FUNCTION_BLOCK "Honeywell_variable_frequency_drives"   // FB29, SCL
{ S7_Optimized_Access := 'TRUE' }
VERSION : 0.1
   VAR_INPUT
      mb_addr : UInt := 255;
   END_VAR
   VAR_IN_OUT
      mb_query : "mb_query";
   END_VAR
   VAR
      sb : "mb_station_block_udt";
      read : Struct
         stw : Struct
            x24 : Bool;
            x25 : Bool;
            x26 : Bool;
            x27 : Bool;
            x28 : Bool;
            x29_control_place : Bool := FALSE;
            x30_control_place : Bool := FALSE;
            x31_control_place : Bool := TRUE;
            x16 : Bool;
            x17 : Bool;
            x18 : Bool;
            x19 : Bool;
            x20 : Bool;
            x21 : Bool;
            x22 : Bool;
            x23 : Bool;
            x08 : Bool;
            x09 : Bool;
            x10 : Bool;
            x11 : Bool;
            x12 : Bool;
            x13 : Bool;
            x14 : Bool;
            x15 : Bool;
            x00_Ready : Bool;
            x01_Running : Bool;
            x02_Counterclockwise : Bool;
            x03_Faulted : Bool;
            x04_Alarm : Bool;
            x05_AtReference : Bool;
            x06_ZeroSpeed : Bool;
            x07_FluxReady : Bool;
         END_STRUCT;
         d1_Output_Frequency : DInt;   // 0,01 Hz
         d2_Motor_Speed : DInt;   // 1 rpm
         d3_Motor_Current : DInt;   // 0,1 A
         d4_Motor_Torque : DInt;   // 0,1 %
         d5_Motor_Power : DInt;   // 0,1 %
         d6_Motor_Voltage : DInt;   // 0,1 V
         d7_DC_link_voltage : DInt;   // 1 V
         d8_Active_Fault_Code : DInt;
      END_STRUCT;
      write : Struct
         ctw : Struct
            x08 : Bool;
            x09 : Bool;
            x10 : Bool;
            x11 : Bool;
            x12 : Bool;
            x13 : Bool;
            x14 : Bool;
            x15 : Bool;
            x00 : Bool;
            x01_start : Bool := TRUE;
            x02_Reverse : Bool;
            x03_Reset_faults : Bool;
            x04 : Bool;
            x05 : Bool;
            x06 : Bool;
            x07 : Bool;
         END_STRUCT;
         __ : Word;
         speed_ref : UInt;   // 0â€¦10000 %
      END_STRUCT;
   END_VAR
BEGIN
   // Honeywell - Variable frequency drives
   // 
   // Web: https://customer.honeywell.com/resources/techlit/
   //      TechLitDocuments/62-0000s/62-0351.pdf

   "mb_station_block_header"(sb := #sb, mb_query := #mb_query);
   #mb_query.mb_addr := #mb_addr;

   #mb_query(mode := #mb_query.c.read.holding_reg,
             data_addr := 2151,
             data_ptr := #read);

   #mb_query(mode := #mb_query.c.write.holding_reg,
             data_addr := 2001,
             data_ptr := #write);

   "mb_station_block_footer"(sb := #sb, mb_query := #mb_query);
END_FUNCTION_BLOCK

// folder: Library/Modbus/Station blocks/Krohne

FUNCTION_BLOCK "Krohne_Optisonic"   // FB34, SCL
{ S7_Optimized_Access := 'TRUE' }
VERSION : 0.1
   VAR_INPUT
      mb_addr : UInt;
   END_VAR
   VAR_IN_OUT
      mb_query : "mb_query";
   END_VAR
   VAR
      sb : "mb_station_block_udt";
      data : Struct
         "Temperature process value" : Real;
         "Dynamic Viscosity at Process conditions" : Real;
         "Density Process" : Real;
         "Flow Process" : Real;
         "Velocity Process" : Real;
         "Speed of Sound" : Real;
      END_STRUCT;
   END_VAR
BEGIN
   // Krohne - Optisonic V6
   // 

   "mb_station_block_header"(sb := #sb,
                             mb_query := #mb_query);
   #mb_query.mb_addr := #mb_addr;

   #mb_query.mode := #mb_query.c.read.holding_reg;
   #mb_query(data_addr := 7050,
             data_ptr := #data);

   "mb_station_block_footer"(sb := #sb,
                             mb_query := #mb_query);
END_FUNCTION_BLOCK

FUNCTION_BLOCK "Krohne_MFC_300"   // FB100, SCL
TITLE = Krohne MFC 300
{ S7_Optimized_Access := 'TRUE' }
AUTHOR : OlaBjornli
FAMILY : modbus
VERSION : 0.1
// Coriolise flow meter
   VAR_INPUT
      mb_addr : UInt;
   END_VAR
   VAR_OUTPUT
      Temperature : Real;   // [degree C]
   END_VAR
   VAR_IN_OUT
      mb_query : "mb_query";
   END_VAR
   VAR
      sb : "mb_station_block_udt";
      read1 : Struct
         "Flow Velocity" : Real;   // [m/s]
         "Volume Flow" : Real;   // [m3/s]
         "Mass Flow" : Real;   // [kg/s]
         Temperature : Real := 273.15;   // [K]
         Density : Real;   // [kg/m3]
         Concentration_1 : Real;
         Concentration_2_or_Diagnosis_3 : Real;
         Concentration_Flow_1 : Real;
         Concentration_Flow_2 : Real;
         Diagnosis_1 : Real;
         Diagnosis_2 : Real;
         Display_Channel_1 : Real;
         Display_Channel_2 : Real;
         Operating_time : Real;   // [s]
      END_STRUCT;
      write1_settings : Struct
         Counter_1_Function : UInt;
         Counter_1_Measurement : UInt;
         Counter_2_Function : UInt;
         Counter_2_Measurement : UInt;
         Counter_3_Function : UInt;
         Counter_3_Measurement : UInt;
      END_STRUCT;
      exec_write : Bool;
   END_VAR
BEGIN
   // Krohne - MFC 300 
   // Flowmeter
   // 
   // Web: http://cdn.krohne.com/dlc/AD_MFC300_Modbus_en_091124_4000744801_R01.pdf
   //
   // #settings :
   //    Counter Function:
   //       1 = Sum Counter
   //       2 = + Counter
   //       3 = - Counter
   //       0 = Off
   //    Counter Measurement:
   //       21 = Volume Flow [m3]
   //       22 = Mass Flow [kg]
   //       27 = Concentration Flow 1
   //       28 = Concentration Flow 2

   "mb_station_block_header"(sb := #sb, mb_query := #mb_query);
   #mb_query.mb_addr := #mb_addr;

   #mb_query(mode := #mb_query.c.mode.read,
             data_addr := 30001, // 30000 + 1 (error in datasheet)
             data_ptr := #read1);
   #Temperature := #read1.Temperature - 273.15;

   // The write query isn't executing continuously in case that will damage eeprom
   IF #exec_write THEN
       #mb_query(mode := #mb_query.c.mode.write,
                 data_addr := 40001, // 40000 + 1,
                 data_ptr := #write1_settings);
       #exec_write := NOT #mb_query.Done;
   END_IF;

   "mb_station_block_footer"(sb := #sb, mb_query := #mb_query);
END_FUNCTION_BLOCK

// folder: Library/Modbus/Station blocks/Mettler

FUNCTION_BLOCK "mettler_toledo_IND560_loadTargetValue"   // FB87, SCL
{ S7_Optimized_Access := 'TRUE' }
VERSION : 0.1
   VAR_INPUT
      iValue : Real;
   END_VAR
   VAR_OUTPUT
      qDone : Bool;
   END_VAR
   VAR_IN_OUT
      "M" : "mettlerToledoInd560Udt";
      sb : "mb_station_block_udt";
   END_VAR
   VAR
      state : Int;
      old_value : Real;
      slot : USInt;
   END_VAR
   VAR CONSTANT
      NONE_AVAILABLE : USInt := 0;
   END_VAR
BEGIN
   // Load target value, for scale 1. Page 143, table B-6

   CASE #state OF

       0:  // Waiting for start.
           #qDone := false;
           #state +=
           BOOL_TO_INT(#old_value <> #iValue);

       1:  // Wait for available msg. slot
           #slot := "reqMsgSlot"(#"M".occupiedMsgSlots);
           #state += BOOL_TO_INT(#slot <> #NONE_AVAILABLE);

       2:  // #1 PLC loads floating point value first
           #"M".writeMsgSlot[#slot].cmd := 0;
           #"M".writeMsgSlot[#slot].data := #iValue;
           #state += 1;
       3:
           #state += BOOL_TO_INT(#"M".queryDone.write);

       4:  // #2 PLC sends command to set target 1 cutoff value 
           #"M".writeMsgSlot[#slot].cmd := 110;
           #state += 1;
       5:
           #state += BOOL_TO_INT(#"M".queryDone.write);

       6:  // #3 IND560 terminal sees new command, loads the value into the target
           //    and ends a return message to indicate the new target value.
           #state +=
           BOOL_TO_INT(#"M".queryDone.read
                       AND #"M".run.cmdAck[#slot] = 1
                       AND #"M".run.PF[#slot] = 13
                       AND #"M".readMsgSlot[#slot].data = #"M".writeMsgSlot[#slot].data);

       7:  // #4  PLC instructs IND560 terminal to start â€œusingâ€ new target value
           #"M".writeMsgSlot[#slot].cmd := 114;
           #state += 1;
       8:
           #state += BOOL_TO_INT(#"M".queryDone.write);

       9:  // #5 IND560 terminal sees new command
           #"M".writeMsgSlot[#slot].cmd := 0;

           #state +=
           BOOL_TO_INT(#"M".queryDone.read
                       AND #"M".run.cmdAck[#slot] = 2
                       AND #"M".run.PF[#slot] = 30
                       AND #"M".readMsgSlot[#slot].data = 0);

       ELSE: // Back to start.
           #"M".occupiedMsgSlots[#slot] := false; // Release msg. slot.
           #state := 0;
           #qDone := true;
           // The start signal should need to be set back false before next
           // exec. else the sequence will start over.
   END_CASE;
   #old_value := #iValue;

   // 
   IF #sb.out.error_comm THEN
       #state := 0;
       IF #slot <> #NONE_AVAILABLE THEN
           #"M".writeMsgSlot[#slot].cmd := 0;
           "releaseMsgSlot"(slot := #slot,
                            mem := #"M".occupiedMsgSlots);
       END_IF;
   END_IF;
END_FUNCTION_BLOCK

FUNCTION_BLOCK "mettler_toledo_IND560"   // FB88, SCL
{ S7_Optimized_Access := 'TRUE' }
VERSION : 0.1
   VAR_IN_OUT
      mb_query : "mb_query";
   END_VAR
   VAR
      mb_addr : UInt := 255;
      sb : "mb_station_block_udt";
      "M" : "mettlerToledoInd560Udt";   // Shared data
      loadTargetValue : "mettler_toledo_IND560_loadTargetValue";
      s : USInt;
   END_VAR
   VAR_TEMP
      c : Int;
   END_VAR
BEGIN
   // Mettler Toledo IND560 - Weighing Terminal

   // WARNING: This SB is just a draft and the block probably include errors !!

   // Necessary settings: ()
   // PLC -> Eth/IP - Modbus TCP -> IP-address
   // PLC -> Eth/IP - Modbus TCP -> Subnet-mask
   // PLC -> Data Format -> Byte order : standard
   // PLC -> Data Format -> Format     : Floating Point 

   // - Modbus tcp:
   //   https://bradysystems.com/wp-content/uploads/2012/10/IND560-PLC-Interface-Manual.pdf
   // - Product overview:
   //   http://www.atsackfillers.mobi/assets/ind560_ug_en_71209396_r04.pdf

   REGION Modbus
       "mb_station_block_header"(sb := #sb,
                                 mb_query := #mb_query);
       #mb_query.mb_addr := #mb_addr;

       #mb_query(mode := #mb_query.c.mode.read,
                 data_addr := 400001,
                 data_ptr := #"M".readMsgSlot,
                 Done => #"M".queryDone.read);

       #mb_query(mode := #mb_query.c.mode.write,
                 data_addr := 401026,
                 data_ptr := #"M".writeMsgSlot,
                 Done => #"M".queryDone.write);

       "mb_station_block_footer"(sb := #sb,
                                 mb_query := #mb_query);
   END_REGION

   REGION Read data-fix     
       // Extract bits in word in to a numbers.
       FOR #c := 1 TO 4 DO
           #"M".run.PF[#c].%X0 := #"M".readMsgSlot[#c].cmdRespons.FP_1;
           #"M".run.PF[#c].%X1 := #"M".readMsgSlot[#c].cmdRespons.FP_2;
           #"M".run.PF[#c].%X2 := #"M".readMsgSlot[#c].cmdRespons.FP_3;
           #"M".run.PF[#c].%X3 := #"M".readMsgSlot[#c].cmdRespons.FP_4;
           #"M".run.PF[#c].%X4 := #"M".readMsgSlot[#c].cmdRespons.FP_5;

           #"M".run.cmdAck[#c].%X0 := #"M".readMsgSlot[#c].cmdRespons.cmdAck1;
           #"M".run.cmdAck[#c].%X1 := #"M".readMsgSlot[#c].cmdRespons.cmdAck2;
       END_FOR;
   END_REGION


   #loadTargetValue(M := #"M",
                    sb := #sb);




   #"M".queryDone.write := false;
   #"M".queryDone.read := false;
END_FUNCTION_BLOCK

FUNCTION "releaseMsgSlot" : Void   // FC17, SCL
{ S7_Optimized_Access := 'TRUE' }
VERSION : 0.1
   VAR_IN_OUT
      slot : USInt;
      mem : Array[*] of Bool;
   END_VAR
   VAR_TEMP
      c : Int;
   END_VAR
BEGIN

   IF #slot <> 0 THEN
       #mem[#slot] := false;
   END_IF;
END_FUNCTION

FUNCTION "reqMsgSlot" : USInt   // FC18, SCL
{ S7_Optimized_Access := 'TRUE' }
VERSION : 0.1
   VAR_IN_OUT
      mem : Array[*] of Bool;
   END_VAR
   VAR_TEMP
      c : Int;
   END_VAR
BEGIN
   // Find first entry inside mem that is false.
   // set the entry to true and return the index. 

   #reqMsgSlot := 0;
   FOR #c := LOWER_BOUND(ARR := #mem, DIM := 1) TO
       UPPER_BOUND(ARR := #mem, DIM := 1)
   DO
       IF NOT #mem[#c] THEN
           #mem[#c] := true;
           #reqMsgSlot := INT_TO_USINT(#c);
           RETURN;
       END_IF;
   END_FOR;
END_FUNCTION

// folder: Library/Modbus/Station blocks/Ponsel mesure

FUNCTION_BLOCK "Ponsel_mesure_Conductivity_C4E"   // FB105, SCL
{ S7_Optimized_Access := 'TRUE' }
VERSION : 0.1
   VAR_INPUT
      mb_addr : UInt := 255;   // 255=broadcast
   END_VAR
   VAR_OUTPUT
      Temperature : Real;   // [degree C]
      Conductivity : Real;   // [uS/cm]
      Salinity : Real;   // [ppt]
      TDS_Kcl : Real;   // [ppm]
      measurement_ok : Bool;
   END_VAR
   VAR_IN_OUT
      mb_query : "mb_query";
   END_VAR
   VAR
      ponsel_mesure : "Ponsel_mesure";
   END_VAR
   VAR_TEMP
      start : Bool;
   END_VAR
BEGIN
   // Ponsel mesure - Conductivity_C4E

   #start := true; // Continuous measurements

   #ponsel_mesure.minimum_measurement_interval := T#1s;
   #ponsel_mesure(mb_addr := #mb_addr,
                  compensate_enable := false,
                  Measurement_ok => #measurement_ok,
                  start_measurement := #start,
                  mb_query := #mb_query);

   #Temperature := #ponsel_mesure.data1.value[0];  // [degree C]
   #Conductivity := #ponsel_mesure.data1.value[1]; // [uS/cm]
   #Salinity := #ponsel_mesure.data1.value[2];     // [ppt]
   #TDS_Kcl := #ponsel_mesure.data1.value[3];      // [ppm]
END_FUNCTION_BLOCK

FUNCTION_BLOCK "Ponsel_mesure_Dissolved_oxygen"   // FB106, SCL
{ S7_Optimized_Access := 'TRUE' }
VERSION : 0.1
   VAR_INPUT
      mb_addr : UInt := 10;   // 255=broadcast
      start : Bool := TRUE;   // (Else use start to init messurements)
      measurement_interval : Time := T#1M;
      compensate_atmospheric_pressure : Real := 1013.0;   // hPa
      compensate_salinity : Real := 0.0;   // ppm
   END_VAR
   VAR_OUTPUT
      Temperature : Real;   // [degree C]
      Oxygen_Sat : Real;   // [%]
      Oxygen_mgl : Real;   // [mg/L]
      Oxygen_ppm : Real;   // [ppm]
      measurement_ok : Bool;
      serial_number : String[32];
   END_VAR
   VAR_IN_OUT
      mb_query : "mb_query";
   END_VAR
   VAR
      ponsel_mesure : "Ponsel_mesure";
   END_VAR
   VAR_TEMP
      start_measurement : Bool;
   END_VAR
BEGIN
   // Aqualabo - Ponsel mesure
   // Dissolved oxygen (OPTOD)
   // 
   // Warning: Each pull for sensor measurement, will reduce the available 
   // life span. Please set the measurement interval to appropriate value.

   #start_measurement := #start; // #measurement_interval will define intervals.

   #ponsel_mesure.minimum_measurement_interval := #measurement_interval;
   #ponsel_mesure.compensate[1] := #compensate_atmospheric_pressure;
   #ponsel_mesure.compensate[2] := #compensate_salinity;
   #ponsel_mesure(mb_addr := #mb_addr,
                  compensate_enable := true,
                  Measurement_ok => #measurement_ok,
                  start_measurement := #start_measurement,
                  mb_query := #mb_query);

   #Temperature := #ponsel_mesure.data1.value[0]; // [degree C]
   #Oxygen_Sat := #ponsel_mesure.data1.value[1];  // [%]
   #Oxygen_mgl := #ponsel_mesure.data1.value[2];  // [mg/l]
   #Oxygen_ppm := #ponsel_mesure.data1.value[3];  // [ppm]

   #serial_number := #ponsel_mesure.data2.serial_number;
END_FUNCTION_BLOCK

// folder: Library/Modbus/Station blocks/Ponsel mesure/Misc

FUNCTION_BLOCK "ponselMessure_ChangeMbAddr"   // FB94, SCL
{ S7_Optimized_Access := 'TRUE' }
VERSION : 0.1
   VAR_INPUT
      current_addr : USInt;
      new_addr : UInt;
      exec : Bool := TRUE;
   END_VAR
   VAR_OUTPUT
      Done : Bool;
      Error : Bool;
   END_VAR
   VAR_IN_OUT
      mb_query : "mb_query";
   END_VAR
   VAR_TEMP
      d : Bool;
      "e" : Bool;
   END_VAR
BEGIN
   IF #new_addr < 1 OR #new_addr > 247
       OR #new_addr = #current_addr
   THEN
       #"e" := TRUE;
   ELSIF #exec THEN
       #mb_query(mb_addr := #current_addr,
                 mode := #mb_query.c.write.holding_reg,
                 data_addr := 16#A3,
                 Done => #d,
                 Error => #"e",
                 data_ptr := #new_addr);
   END_IF;
   #Done := #d;
   #Error := #"e";
END_FUNCTION_BLOCK

FUNCTION_BLOCK "Ponsel_mesure"   // FB107, SCL
{ S7_Optimized_Access := 'TRUE' }
VERSION : 0.1
   VAR_INPUT
      mb_addr : UInt;
      minimum_measurement_interval : Time := T#1M;
      compensate_enable : Bool;
      compensate : Array[1..2] of Real;
   END_VAR
   VAR_OUTPUT
      Measurement_ok : Bool;
   END_VAR
   VAR_IN_OUT
      mb_query : "mb_query";
      start_measurement : Bool;
   END_VAR
   VAR
      sb : "mb_station_block_udt";
      QueryCnt : UDInt;
      data1 : Struct
         value : Array[0..4] of Real;
         compensate_temperature : Real;
         compensate : Array[1..2] of Real;
         _ : Word;
         status : Array[0..4] of Struct
            x08_StmGamme0 : Bool;
            x09_StmGamme1 : Bool;
            x10_StmGamme2 : Bool;
            x11 : Bool;
            x12 : Bool;
            x13 : Bool;
            x14 : Bool;
            x15 : Bool;
            x00_Stm0 : Bool;
            x01_Stm1 : Bool;
            x02_Stm2 : Bool;
            x03_StmTemp : Bool;   // At least one parameter coefficient uses a temporary calibration standard (configuration during calibration)
            x04_StmHF : Bool;   // At least one parameter coefficient is outside calibration limits
            x05_StmCU : Bool;   // All parameter coefficients use default coefficient
            x06_StmHIST : Bool;   // All parameter coefficients use history coefficient
            x07_StmME : Bool;   // Dry weight is missing in at least one parameter coefficient (measurement under way)
         END_STRUCT;
         Compensates_3 : Real;
      END_STRUCT;
      data2 : Struct
         Description : String[30];
         serial_number : String[32];   // (addr 0x0D10)
         Software_version : Word;   // Heavy Weight: Major version and Light Weight: Minor Version.
         Hardware_version : Word;   // Heavy Weight: Major version and Light Weight: Minor Version.
      END_STRUCT;
      api : Struct
         idle : Bool;
         wait : Bool;
         interval : Time;
      END_STRUCT;
      _ : Bool;   // Internal variables bellow.
      state : Int;
      "timer" : TON_TIME;
      timer_in : Bool;
      timer_q : Bool;
      first_scan : Bool := TRUE;
      wait_time : UInt;
   END_VAR
   VAR_TEMP
      "word" : Word;
      c : Int;
      error : Bool;
      tIdle : Bool;
      pt : Time;
   END_VAR
BEGIN
   // Aqualabo - Ponsel mesure
   // Dissolved oxygen (OPTOD), Conductivity (C4E, CTZ), pH_Redox, Turbi    
   // 
   // - Warning: For the oxygen sensor each pull for sensor measurement,
   //   will use of the available life span. Please set the measurement
   //   interval to appropriate value.
   // - Continuous assign true to start_measurement, to continuous do
   //   meassurements. #minimum_measurement_interval wil still restrict
   //   the interval time.
   // - https://en.aqualabo.fr/userfiles/doc/User%20Manual%20Oxygen%20Optical%20digital%20sensor%20OPTOD.pdf

   "mb_station_block_header"(sb := #sb,
                             mb_query := #mb_query);
   #mb_query.mb_addr := #mb_addr;
   #mb_query.mode := #mb_query.c.read.holding_reg;

   #"timer"(IN := #timer_in,
          PT := #"timer".PT,
          Q => #timer_q);
   #timer_in := false;

   IF #sb.out.error_comm THEN // If communication error
       #state := 0;
       #Measurement_ok := false;
       #timer_in := true;  // Continue run the timer.
   ELSE
       CASE #state OF
           1:  // Compensate: Salinity, barometric pressure, temperature, etc.
               IF #compensate_enable THEN
                   #mb_query(mode := #mb_query.c.write.holding_reg,
                             data_addr := 16#5f,
                             data_ptr := #compensate);
                   #state += BOOL_TO_INT(#mb_query.Done);
               ELSE
                   #state += 1;
               END_IF;
           2:  // Read wait-time (Used later in state 4)
               #mb_query(data_addr := 16#A4,
                         data_ptr := #wait_time);
               #state += BOOL_TO_INT(#mb_query.Done);
           3:  // Start all meassurements.
               #"word" := 16#0f;
               #mb_query(mode := #mb_query.c.write.holding_reg,
                         data_addr := 16#01,
                         data_ptr := #"word");
               #state += BOOL_TO_INT(#mb_query.Done);
           4:  // Timer (Wait while sensor is obtaining measurements)
               #timer_in := true;
               PRESET_TIMER(TIMER := #"timer",
                            PT := MAX(IN1 := T_CONV(#wait_time),
                                      IN2 := T#1s)); // No less then 1s.
               #state += BOOL_TO_INT(#timer_q);
           5:  // Get data.
               #mb_query(data_addr := 16#0053,
                         data_ptr := #data1);
               // All measurements ok ?
               FOR #c := 0 TO 4 DO
                   #error := #error
                   OR #data1.status[#c].x00_Stm0
                   OR #data1.status[#c].x01_Stm1
                   OR #data1.status[#c].x02_Stm2;
               END_FOR;
               #Measurement_ok := NOT #error;
               IF #mb_query.Done THEN
                   // #start_measurement need to be assigned
                   // true again to start a new messurement.
                   #start_measurement := false;
                   #state := 0;
                   #QueryCnt += 1;
               END_IF;
           ELSE
               #tIdle := true;
               #timer_in := true;
               #pt := SEL(G := #api.interval = T#0s,
                          IN0 := #api.interval,
                          IN1 := #minimum_measurement_interval);
               PRESET_TIMER(PT := #pt,
                            TIMER := #"timer");

               #state := BOOL_TO_INT
               (NOT #api.wait AND // #api.wait may be set by other
                // function blocks to  halt the messurements.
                #start_measurement AND (
                (* *)#timer_q // Interval controlled
                (* *)OR #first_scan)); // At statup a messurement
               // is done as fast as possible.
       END_CASE;
   END_IF;
   // #wait is a API, for other blocks to stop the messurements,
   // #idle tells other blocks that no messurement is in progress.


   IF #sb.out.error_comm
       OR #api.idle AND NOT #api.wait
   THEN
       // Description, Serial number, sw and hw version.
       #mb_query(data_addr := 3327,
                 data_ptr := #data2);
   END_IF;

   "mb_station_block_footer"(sb := #sb,
                             mb_query := #mb_query);

   #api.idle := #tIdle;
   #api.wait := false;
   #api.interval := T#0s;
   #first_scan := false;

   (* 
   Units:
   ---------------
   value0: Temperature
                         value1:                    value2:                    value3:       
   OPTOD (oxygen)    :   Oxygen [%Sat]              Oxygen [mg/l]              Oxygen [ppm]
   Turbi             :   Nephelo turbidity [NTU]    Nephelo turbidity [FNU]    TU turbidity [mg/L]
   pH_Redox          :   pH                         Redox [mV]
   conductivity_C4E  :   Conductivity C4E [uS/cm]   Salinity [ppt]             TDS - Kcl [ppm]
   Conductivity_CTZ  :   Conductivity CTZ [mS/cm]   Salinity [g/Kg]            Conductivity CTZ [mS/cm] 
                                                                               without temperature compensation                                                                  
   OPTOD: (Dissolved oxygen)
   Compensates[1]: Atmospheric pressure [hPa], default 1013 hPa
   Compensates[2]: Salinity [ppt], default 0 ppt


   Wiring: 
   Red     Wiring diagram V+
   black   Wiring diagram V-
   Green   B+ RS-485  (Siemens A)
   White   A- RS-485  (Siemens B)
   Blue    SDI-12

   Default settings:
   Buad: 9600
   Parity: none
   Modbus address: 10


   StmX:
   000: Measurement OK
   001: Measurement OK, but out of specifications
   010: Measurement OK with INFO 1 (See datasheet)
   011: Measurement OK with INFO 2 (See datasheet)
   100: Measurement impossible, out of specifications
   101: Measurement impossible with INFO 3 (See datasheet)
   110: Measurement impossible with INFO 4 (See datasheet)
   111: measurement under way (not yet available)

   StmGamme:       
   001: measurement used range 1
   010: measurement used range 2
   011: measurement used range 3
   100: measurement used range 4

   *)
END_FUNCTION_BLOCK

// folder: Library/Modbus/Station blocks/Produal

FUNCTION_BLOCK "produal_KLH_M"   // FB42, SCL
{ S7_Optimized_Access := 'TRUE' }
VERSION : 0.1
   VAR_INPUT
      mb_addr : USInt;
   END_VAR
   VAR_OUTPUT
      temperature : Real;
      humidity : Real;
      potentiometer : Real;
   END_VAR
   VAR_IN_OUT
      mb_query : "mb_query";
   END_VAR
   VAR
      sb : "mb_station_block_udt";
      write1_calibration : Struct
         temp_offset : Int;
         humidity_offset : Int;
      END_STRUCT;
      read1 : Struct
         temperature : Int;
         humidity : UInt;
         y : Array[1..4] of UInt;
         potentiometer : Int;   // %
      END_STRUCT;
   END_VAR
BEGIN
   // Produal - KLH-M
   // Product number: 1132600
   // http://www.produal.com/shop/web_humidity_transmitters/sku-1132600

   "mb_station_block_header"(sb := #sb, mb_query := #mb_query);
   #mb_query.mb_addr := #mb_addr;

   #mb_query(mode := #mb_query.c.mode.read,
             data_addr := 30001,
             data_ptr := #read1);

   #mb_query(mode := #mb_query.c.mode.write,
             data_addr := 40006,
             data_ptr := #write1_calibration); // temp. and humidity  

   "mb_station_block_footer"(sb := #sb, mb_query := #mb_query);

   #temperature := INT_TO_REAL(#read1.temperature) * 0.1;
   #humidity := UINT_TO_REAL(#read1.humidity); // 0-100%
   #potentiometer := INT_TO_REAL(#read1.potentiometer) * 0.1;
END_FUNCTION_BLOCK

FUNCTION_BLOCK "produal_TEHR_M"   // FB43, SCL
{ S7_Optimized_Access := 'TRUE' }
VERSION : 0.1
   VAR_INPUT
      mb_addr : USInt;
      calibration_offset : Int;   // mbar
   END_VAR
   VAR_OUTPUT
      temperature : Real;   // Â°C
      analogue_output : Real;   // V
      potentiometer : Real;   // %
   END_VAR
   VAR_IN_OUT
      mb_query : "mb_query";
   END_VAR
   VAR
      sb : "mb_station_block_udt";
      r1 : Struct
         temperature : Int;
         analogue_output : UInt;
         potentiometer : Int;
      END_STRUCT;
   END_VAR
BEGIN
   // Produal - TEHR-M - Temperatur transmitter.
   // Product: 117Z190 - Pt1000 EN 60751/B
   // http://www.produal.com/shop/web_bus_temperature_transmitters/
   // sku-117Z190?hiddenAttributes_sensor_output=sensor_output_modbus&saf=true

   "mb_station_block_header"(sb := #sb,
                             mb_query := #mb_query);
   #mb_query.mb_addr := #mb_addr;

   #mb_query(mode := #mb_query.c.mode.read,
             data_addr := 30001,
             data_ptr := #r1);

   #mb_query(mode := #mb_query.c.mode.write,
             data_addr := 40001,
             data_ptr := #calibration_offset);

   "mb_station_block_footer"(sb := #sb,
                             mb_query := #mb_query);

   #temperature := INT_TO_REAL(#r1.temperature) * 0.1;
   #analogue_output := UINT_TO_REAL(#r1.analogue_output);
   #potentiometer := INT_TO_REAL(#r1.potentiometer) * 0.1;
END_FUNCTION_BLOCK

// folder: Library/Modbus/Station blocks/Scandinavian Electric

FUNCTION_BLOCK "Scandinavian_electric_CEM M-RS485"   // FB45, SCL
{ S7_Optimized_Access := 'TRUE' }
VERSION : 0.1
   VAR_INPUT
      mb_addr : UInt;
   END_VAR
   VAR_IN_OUT
      mb_query : "mb_query";
   END_VAR
   VAR
      sb : "mb_station_block_udt";
      read1 : Struct
         "Imported active energy" : UDInt;
         "Exported active energy" : UDInt;
         "Q1 Reactive energy" : UDInt;
         "Q2 Reactive energy" : UDInt;
         "Q3 Reactive energy" : UDInt;
         "Q4 Reactive energy" : UDInt;
      END_STRUCT;
      read2 : Struct
         "Partial imported active energy" : UDInt;
         "Partial exported active energy" : UDInt;
         "Q1 partial reactive energy" : UDInt;
         "Q2 partial reactive energy" : UDInt;
         "Q3 partial reactive energy" : UDInt;
         "Q4 partial reactive energy" : UDInt;
      END_STRUCT;
      serial_number : UDInt;
   END_VAR
BEGIN
   // Scandinavian Electric - Circutor - CEM M-RS485
   // Modbus interface for CEM energy meters

   // - Note: Only no parity.
   // - http://scel.no/produkter/energimaling_/_3_fase_malere/
   //   content/text_432575b2-b97f-4834-84d7-3fb83a2fdd40/1442214133237/
   //   cem_m_rs485.pdf
   // - (M014B01-03-14A)

   "mb_station_block_header"(sb := #sb, mb_query := #mb_query);
   #mb_query.mb_addr := #mb_addr;

   #mb_query.mode := #mb_query.c.read.holding_reg;
   #mb_query(data_addr := 16#0000, data_ptr := #read1);
   #mb_query(data_addr := 16#0030, data_ptr := #read2);
   #mb_query(data_addr := 16#2710, data_ptr := #serial_number);

   "mb_station_block_footer"(sb := #sb, mb_query := #mb_query);
END_FUNCTION_BLOCK

FUNCTION_BLOCK "Scandinavian_electric_Circutor_CBS"   // FB46, SCL
{ S7_Optimized_Access := 'TRUE' }
VERSION : 0.1
   VAR_INPUT
      mb_addr : UInt;
   END_VAR
   VAR_IN_OUT
      mb_query : "mb_query";
   END_VAR
   VAR
      sb : "mb_station_block_udt";
      data : Struct
         current : Array[1..8] of UInt;   // [mA]
         outputs : Array[1..8] of UInt;   // 0=Normal, 1=Pre-alarm, 2=Aktivert, 3=LÃ¥st
         pre_alarm_relay : UInt;
      END_STRUCT;
      limits : Array[1..8] of UInt;   // [mA]
   END_VAR
BEGIN
   // Scandinavian Electric - Circutor - CBS-8
   // 
   // - http://scel.no/produkter/jordfeilovervaking/
   //   varsler_panel_og_scanningsystem/content_2/
   //   text_8e3609e0-231d-4dfc-80a4-71ee43eee1af/1409662445698/cbs8.pdf

   "mb_station_block_header"(sb := #sb, mb_query := #mb_query);
   #mb_query.mb_addr := #mb_addr;

   #mb_query.mode := #mb_query.c.write.holding_reg;
   #mb_query(data_addr := 13, data_ptr := #limits);

   #mb_query.mode := #mb_query.c.read.holding_reg;
   #mb_query(data_addr := 2, data_ptr := #data);

   "mb_station_block_footer"(sb := #sb, mb_query := #mb_query);
END_FUNCTION_BLOCK

// folder: Library/Modbus/Station blocks/Schneider

FUNCTION_BLOCK "Schneider_ATV6xx"   // FB47, SCL
{ S7_Optimized_Access := 'TRUE' }
VERSION : 0.1
   VAR_INPUT
      mb_addr : USInt;
      ref_freq : Real;
   END_VAR
   VAR_IN_OUT
      mb_query : "mb_query";
   END_VAR
   VAR
      sb : "mb_station_block_udt";
      write1 : Struct
         cmd_reg : Struct
            x08_halt : Bool;
            x09 : Bool;
            x10 : Bool;
            x11_Reverse : Bool;
            x12 : Bool;
            x13 : Bool;
            x14 : Bool;
            x15 : Bool;
            x00_switch_on : Bool := TRUE;
            x01_enable_voltage : Bool := TRUE;
            x02_quick_stop : Bool;
            x03_Run : Bool;
            x04 : Bool;
            x05 : Bool;
            x06 : Bool;
            x07_fault_reset : Bool;
         END_STRUCT;
         ref_freq : Int;
      END_STRUCT;
      read1 : Struct
         status : Struct   // ETA
            x08 : Bool;
            x09_remote : Bool;   // Command or reference value via fieldbus
            x10_on_target : Bool;   // Reference value reached
            x11_ref_outside_lim : Bool;   // Reference value outside limits
            x12 : Bool;
            x13 : Bool;
            x14_stop_key : Bool;   // Manufacturer-specific Stop via STOP key
            x15_reverse : Bool;   // Manufacturer-specific
            x00_awaiting_power_stage_supply : Bool;
            x01_ready : Bool;
            x02_running : Bool;
            x03_fault : Bool;
            x04_power_stage_supply_present : Bool;
            x05_quick_stop : Bool;
            x06_power_stage_supply_disabled : Bool;
            x07_warning : Bool;
         END_STRUCT;
         output_frequency : Int;   // RFR
         frequency_reference_before_ramp : Int;   // FRH
         motor_current : Int;   // LCR
         motor_torque : Int;   // OTR
         ext_status_word : Word;
         mains_voltage : Int;   // ULN
         motor_voltage : Int;   // UOP
         drive_thermal_state : Int;   // THD
      END_STRUCT;
   END_VAR
BEGIN
   // Schneider - ATV6xx (EAV94279)
   //  
   // - http://www2.schneider-electric.com/resources/sites/SCHNEIDER_ELECTRIC/
   //   content/live/FAQS/275000/FA275868/en_US/
   //   Process%20drive%20communication%20parameters.xlsx
   // - https://profsector.com/media/catalogs/56e3af69500ef.pdf
   // - https://download.schneider-electric.com/
   //   files?p_enDocType=User+guide&p_File_Id=5470508810&
   //   p_File_Name=ATV600_EthernetIP_Modbus_TCP_Manual_EN_EAV6
   //   4328_02.pdf&p_Reference=EAV64328

   #write1.ref_freq := REAL_TO_INT(#ref_freq * 10);
   #write1.cmd_reg.x00_switch_on := #write1.cmd_reg.x03_Run := #ref_freq <> 0;

   "mb_station_block_header"(sb := #sb, mb_query := #mb_query);
   #mb_query.mb_addr := #mb_addr;

   #mb_query.mode := #mb_query.c.write.holding_reg;
   #mb_query(data_addr := 8501, data_ptr := #write1);

   #mb_query.mode := #mb_query.c.read.holding_reg;
   #mb_query(data_addr := 3201, data_ptr := #read1);

   "mb_station_block_footer"(sb := #sb, mb_query := #mb_query);
END_FUNCTION_BLOCK

FUNCTION_BLOCK "Schneider_PM556x_series"   // FB48, SCL
{ S7_Optimized_Access := 'TRUE' }
VERSION : 0.1
   VAR_INPUT
      mb_addr : UInt;
   END_VAR
   VAR_IN_OUT
      mb_query : "mb_query";
   END_VAR
   VAR
      sb : "mb_station_block_udt";
      Accumulated_Energy : Struct
         "Active Energy Delivered (Into Load)" : Real;   // kWh
         "Active Energy Received (Out of Load)" : Real;   // kWh
         "Active Energy Delivered + Received" : Real;   // kWh
         "Active Energy Delivered- Received" : Real;   // kWh
         "Reactive Energy Delivered" : Real;   // kVARh
         "Reactive Energy Received" : Real;   // kVARh
         "Reactive Energy Delivered + Received" : Real;   // kVARh
         "Reactive Energy Delivered - Received" : Real;   // kVARh
         "Apparent Energy Delivered" : Real;   // kVAh
         "Apparent Energy Received" : Real;   // kVAh
         "Apparent Energy Delivered + Received" : Real;   // kVAh
         "Apparent Energy Delivered - Received" : Real;   // kVAh
      END_STRUCT;
      data1 : Struct
         Current : Array[1..3] of Real;   // A
         "Current N" : Real;   // A
         "Current G" : Real;   // A
         "Current Avg" : Real;   // A
         "Current Unbalance" : Array[1..3] of Real;   // %
         "Current Unbalance Worst" : Real;   // %
         "Voltage L-L" : Array[1..3] of Real;   // V
         "Voltage L-L Avg" : Real;   // V
         "Voltage L-N" : Array[1..3] of Real;   // V
         "Voltage L-N Avg" : Real;   // V
         "Voltage Unbalance L-L" : Array[1..3] of Real;   // %
         "Voltage Unbalance L-L Worst" : Real;   // %
         "Voltage Unbalance L-N" : Array[1..3] of Real;   // %
         "Voltage Unbalance L-N Worst" : Real;   // %
      END_STRUCT;
      Power : Struct
         "Active Power" : Array[1..3] of Real;   // kW
         "Active Power Total" : Real;   // kW
         "Reactive Power" : Array[1..3] of Real;   // kVAR
         "Reactive Power Total" : Real;   // kVAR
         "Apparent Power" : Array[1..3] of Real;   // kVA
         "Apparent Power Total" : Real;   // kVA
         "Power Factor" : Array[1..3] of Real;   // ---
         "Power Factor Total" : Real;   // ---
         "Displacement Power Factor" : Array[1..3] of Real;   // ---
         "Displacement Power Factor Total" : Real;   // ---
      END_STRUCT;
      PF : Struct
         "Power Factor" : Array[1..3] of Real;
         "Power Factor Total" : Real;
         "Displacement Power Factor" : Array[1..3] of Real;
         "Displacement Power Factor Total" : Real;
      END_STRUCT;
      Frequency : Real;   // Hz
   END_VAR
   VAR_TEMP
      c : Int;
      t1 : Real;
      t2 : Real;
   END_VAR
BEGIN
   // Schneider Electric - PM5560, PM5563, PM5563RD
   // 
   // https://www.schneider-electric.com/en/faqs/FA234017/

   "mb_station_block_header"(sb := #sb, mb_query := #mb_query);
   #mb_query.mb_addr := #mb_addr;

   #mb_query.mode := #mb_query.c.read.holding_reg;
   #mb_query(data_addr := 2700, data_ptr := #Accumulated_Energy);
   #mb_query(data_addr := 3000, data_ptr := #data1);
   #mb_query(data_addr := 3054, data_ptr := #Power);
   #mb_query(data_addr := 3110, data_ptr := #Frequency);

   "mb_station_block_footer"(sb := #sb, mb_query := #mb_query);

   FOR #c := 1 TO 8 DO
       (* Power factor values are specially encoded floating point 
       values. Angle of complex power = power factor register value
       0° = 1, 90° = 0,  180° = -1,  270° = 2,  Q1: 0 < x < 1
       Q2: -2 < x < -1,  Q3:  -1 < x < 0,   Q4: 1 < x < 2  *)
       CASE #c OF
           1..3: #t1 := #Power."Power Factor"[#c];
           4:    #t1 := #Power."Power Factor Total";
           5..7: #t1 := #Power."Displacement Power Factor"[#c - 4];
           8:    #t1 := #Power."Displacement Power Factor Total";
       END_CASE;
       IF #t1 > 1 THEN // PF is leading
           #t2 := 2 - #t1;
       ELSIF #t1 < -1 THEN // PF is leading
           #t2 := -2 - #t1;
       ELSE            // ABS(#t1) = 1 -> PF is at unity
           #t2 := #t1; // else -> PF is lagging
       END_IF;
       CASE #c OF
           1..3: #PF."Power Factor"[#c] := #t2;
           4:    #PF."Power Factor Total" := #t2;
           5..7: #PF."Displacement Power Factor"[#c - 4] := #t2;
           8:    #PF."Displacement Power Factor Total" := #t2;
       END_CASE;
   END_FOR;
END_FUNCTION_BLOCK

FUNCTION_BLOCK "Schneider_PM1000_series"   // FB49, SCL
TITLE = Schneider Electric - PM1000 Series Power Meters
{ S7_Optimized_Access := 'TRUE' }
VERSION : 0.1
   VAR_INPUT
      mb_addr : UInt;
   END_VAR
   VAR_OUTPUT
      all : Struct
         apparent_power : Real;
         active_power : Real;
         reactive_power : Real;
         power_factor : Real;
         voltage_L_L : Real;
         voltage_L_N : Real;
         current : Real;
      END_STRUCT;
      phase : Array[1..3] of Struct
         apparent_power : Real;
         active_power : Real;
         reactive_power : Real;
         power_factor : Real;
         voltage_L_L : Real;
         voltage_L_N : Real;
         current : Real;
      END_STRUCT;
   END_VAR
   VAR_IN_OUT
      mb_query : "mb_query";
   END_VAR
   VAR
      sb : "mb_station_block_udt";
   END_VAR
   VAR_TEMP
      tAll : Struct
         apparent_power : DWord;
         active_power : DWord;
         reactive_power : DWord;
         power_factor : DWord;
         voltage_L_L : DWord;
         voltage_L_N : DWord;
         current : DWord;
      END_STRUCT;
      tPhase : Array[1..3] of Struct
         apparent_power : DWord;
         active_power : DWord;
         reactive_power : DWord;
         power_factor : DWord;
         voltage_L_L : DWord;
         voltage_L_N : DWord;
         current : DWord;
      END_STRUCT;
      c : Int;
   END_VAR
BEGIN
   // Schneider Electric - PowerLogic - PM1000 Series Power Meters
   //  - PM1200
   // 
   // http://static.schneider-electric.us/docs/Power%20Management/
   // PowerLogic%20Products/Metering/PM1200%20power%20meter/
   // PLSED309039EN_PM1000_UG.pdf

   "mb_station_block_header"(sb := #sb,
                             mb_query := #mb_query);
   #mb_query.mb_addr := #mb_addr;

   #mb_query.mode := #mb_query.c.read.holding_reg;

   #mb_query(data_addr := 3901,
             data_ptr := #tAll);
   IF #mb_query.Done THEN
       #all.apparent_power := DWORD_TO_REAL(SWAP(#tAll.apparent_power));
       #all.active_power := DWORD_TO_REAL(SWAP(#tAll.active_power));
       #all.reactive_power := DWORD_TO_REAL(SWAP(#tAll.reactive_power));
       #all.power_factor := DWORD_TO_REAL(SWAP(#tAll.power_factor));
       #all.voltage_L_L := DWORD_TO_REAL(SWAP(#tAll.voltage_L_L));
       #all.voltage_L_N := DWORD_TO_REAL(SWAP(#tAll.voltage_L_N));
       #all.current := DWORD_TO_REAL(SWAP(#tAll.current));
   END_IF;

   FOR #c := 1 TO 3 DO
       CASE #c OF
           1:
               #mb_query.data_addr := 3917;
           2:
               #mb_query.data_addr := 3931;
           3:
               #mb_query.data_addr := 3945;
       END_CASE;
       #mb_query(data_ptr := #tPhase[#c]);
       IF #mb_query.Done THEN
           #phase[#c].apparent_power := DWORD_TO_REAL(SWAP(#tPhase[#c].apparent_power));
           #phase[#c].active_power := DWORD_TO_REAL(SWAP(#tPhase[#c].active_power));
           #phase[#c].reactive_power := DWORD_TO_REAL(SWAP(#tPhase[#c].reactive_power));
           #phase[#c].power_factor := DWORD_TO_REAL(SWAP(#tPhase[#c].power_factor));
           #phase[#c].voltage_L_L := DWORD_TO_REAL(SWAP(#tPhase[#c].voltage_L_L));
           #phase[#c].voltage_L_N := DWORD_TO_REAL(SWAP(#tPhase[#c].voltage_L_N));
           #phase[#c].current := DWORD_TO_REAL(SWAP(#tPhase[#c].current));
       END_IF;
   END_FOR;

   "mb_station_block_footer"(sb := #sb,
                             mb_query := #mb_query);
END_FUNCTION_BLOCK

FUNCTION_BLOCK "Schneider_power_meter_750"   // FB50, SCL
{ S7_Optimized_Access := 'TRUE' }
VERSION : 0.1
   VAR_INPUT
      mb_addr : UInt;
   END_VAR
   VAR_IN_OUT
      mb_query : "mb_query";
   END_VAR
   VAR
      sb : "mb_station_block_udt";
      data1 : Struct
         "Real Energy, Total" : Real;   // kWh
         "Apparent Energy,Tota" : Real;   // kVAh
         "Reactive Energy,Tota" : Real;   // kVARh
         "Real Power, Total" : Real;   // kW
         "Apparent Power, Total" : Real;   // kVA
         "Reactive Power, Total" : Real;   // kVAR
         "Power Factor, Total" : Real;
         "Voltage, L-L, 3PAverage" : Real;   // Volt
         "Voltage, L-N, 3PAverage" : Real;   // Volt
         "Current, 3P Average" : Real;   // Amp
         Frequency : Real;
      END_STRUCT;
      data2 : Struct
         Current : Array[1..3] of Real;
         Current_N : Real;
      END_STRUCT;
      data3 : Struct
         Voltage_L_L : Array[1..3] of Real;   // [V] 1:L1-L2, 2:L2-L3, 3:L3-L1
         Voltage_L_N : Array[1..3] of Real;   // [V]
         "Real Power" : Array[1..3] of Real;   // kW
         "Apparent Power" : Array[1..3] of Real;   // kVA
         "Reactive Power" : Array[1..3] of Real;   // kVAR
      END_STRUCT;
   END_VAR
BEGIN
   // Schneider - Power Meter 750
   // 63230-507-201A1 - 03/2007
   // 
   // Web: https://www.ccontrols.com/support/dp/SchneiderElectricPowerMeter750.pdf

   "mb_station_block_header"(sb := #sb,
                             mb_query := #mb_query);
   #mb_query.mb_addr := #mb_addr;

   #mb_query.mode := #mb_query.c.read.holding_reg;
   #mb_query(data_addr := 1000,
             data_ptr := #data1);
   #mb_query(data_addr := 1034,
             data_ptr := #data2);
   #mb_query(data_addr := 1054,
             data_ptr := #data3);

   "mb_station_block_footer"(sb := #sb,
                             mb_query := #mb_query);
END_FUNCTION_BLOCK

FUNCTION_BLOCK "Schneider_SCADAPack_4000"   // FB51, SCL
{ S7_Optimized_Access := 'TRUE' }
VERSION : 0.1
   VAR_INPUT
      mb_addr : UInt;
   END_VAR
   VAR_IN_OUT
      mb_query : "mb_query";
   END_VAR
   VAR
      sb : "mb_station_block_udt";
      data : Array[1..3] of Int;
      setting : Array[1..3] of Int;
   END_VAR
BEGIN
   // Schneider - SCADAPack 4000 
   // Models 4012, 4032 and 4102 - Transmitters
   // 
   // Web: https://s3.amazonaws.com/cdn.freshdesk.com/data/helpdesk/
   // attachments/production/5013914262/original/
   // SCADAPack_4000_Series_Transmitters.pdf?
   // X-Amz-Algorithm=AWS4-HMAC-SHA256&X-Amz-Credential=
   // AKIAJ2JSYZ7O3I4JO6DA%2F20170919%2Fus-east-1%2Fs3%2Faws4_
   // request&X-Amz-Date=20170919T163931Z&X-Amz-Expires=300&X-Amz-
   // Signature=a206005821114e23f4a38162afdf9d14bd82209c246a378f18
   // 9af628740a1509&X-Amz-SignedHeaders=Host&response-content-type=
   // application%2Fpdf

   "mb_station_block_header"(sb := #sb, mb_query := #mb_query);
   #mb_query.mb_addr := #mb_addr;

   #mb_query.mode := #mb_query.c.mode.read;
   #mb_query(data_addr := 40116, data_ptr := #data);

   #mb_query.mode := #mb_query.c.mode.write;
   #mb_query(data_addr := 40060, data_ptr := #setting);

   "mb_station_block_footer"(sb := #sb, mb_query := #mb_query);

   (*
   Setting:

   value[1] and value[2]
   ------------------
   2 = Pascal (Pa)
   3 = kiloPascal (kPa)
   4 = megaPascal (MPa)
   5 = pounds per square inch (psi)
   6 = inches of water at 68 F
   7 = ftH2O
   8 = atm
   9 = bar
   10 = kg/cm2
   11 = g/cm2
   12 = cmHg
   13 = mmHg
   14 = torr
   15 = mH2O
   16 = cmH2O
   17 = mmH2O
   18 = inHg
   19 = mbar


   value[3]
   ------------------
   20 = degrees Celsius (ï‚°C)
   21 = degrees Fahrenheit (ï‚°F)
   22 = degrees Kelvin (K)
   23 = degrees Rankine(R)

   *)
END_FUNCTION_BLOCK

FUNCTION_BLOCK "Telemecanique_Schneider_Altivar_21_inverter"   // FB71, SCL
{ S7_Optimized_Access := 'TRUE' }
VERSION : 0.1
   VAR_INPUT
      mb_addr : UInt;
      ref : Real;
      acceleration_time : Real;
   END_VAR
   VAR_IN_OUT
      mb_query : "mb_query";
   END_VAR
   VAR
      sb : "mb_station_block_udt";
      data : Struct
         Output_current : Real;
         Voltage_DC_bus : Real;
         Output_frequency : Real;
      END_STRUCT;
      read1 : Struct   // 16#fd00
         Output_frequency : Word;
         stat : Struct
            x08 : Bool;
            x09_Reverse : Bool;
            x10_Run : Bool;
            x11_Coast_stop : Bool;
            x12_Emergency_stop : Bool;
            x13_Standby_ST_ON : Bool;   // Standby: Initialization completed, not failure stop status, not alarm stop status (MOFF, LL forced stop or forced stop due to a momentary power failure), ST=ON, and RUN=ON
            x14_Standby : Bool;   // Standby: Initialization completed, not failure stop status, and not alarm stop status (MOFF, LL forced stop or forced stop due to a momentary power failure)
            x15_Local : Bool;
            x00_Failure_FL : Bool;
            x01_Failure : Bool;
            x02_Alarm : Bool;
            x03_Main_circuit_undervoltage : Bool;
            x04_THR_2 : Bool;   // THR1: PT=set value, vL, vb, Thr - THR2: PT=0, F170, F172, F173
            x05_PI_control_OFF : Bool;
            x06_Acceleration2_deceleration2 : Bool;
            x07_DC_braking : Bool;
         END_STRUCT;
      END_STRUCT;
      read2 : Struct   // 16#fe45
         Command_mode : UInt;   // 0:Terminal board, 1:Operation panel, 2:Serial
         Setpoint_mode : UInt;   // 1 VIA, 2 VIB, 3 Operation panel, 4 Serial, 5 TB up down frequency, 255 Preset speed operation
      END_STRUCT;
      read3_alarm : Struct   // 16#fe91
         x08_Over_torque : Bool;
         x09_Cumulative_operation_hours : Bool;
         x10 : Bool;
         x11 : Bool;
         x12 : Bool;
         "x13_Main circuit_undervoltage" : Bool;   // same as MS-relay status
         x14_Decelerating_stopping : Bool;   // Related: F256 setting. At the time of the instant blackout, Forced deceleration/stop
         x15_Decelerating_stopping : Bool;   // Related: F302 setting. An automatic stop during the lower limit frequency continuance
         x00_Overcurrent : Bool;
         x01_Inverter_overload : Bool;
         x02_Motor_overload : Bool;
         x03_Overheat : Bool;
         x04_Overvoltage : Bool;
         x05_Main_circuit_undervoltage : Bool;
         x06 : Bool;
         x07_Undercurrent : Bool;
      END_STRUCT;
      read4_alarm2 : Struct   // 16#fe79
         x08 : Bool;
         x09 : Bool;
         x10 : Bool;
         x11 : Bool;
         x12 : Bool;
         x13 : Bool;
         x14 : Bool;
         x15 : Bool;
         x00_Fan_life_alarm : Bool;
         x01_Circuit_board_life : Bool;
         x02_Main_circuit_capacitor_life : Bool;
         x03_User_set_alarm : Bool;
         x04 : Bool;
         x05 : Bool;
         x06 : Bool;
         x07 : Bool;
      END_STRUCT;
      read5_trip_code : UInt;   // 16#fc90
      write1 : Struct
         cmd : Struct
            x08 : Bool;
            x09_Reverse : Bool;
            x10_Run : Bool;
            x11_Coast_stop : Bool;
            x12_Emergency_stop : Bool;
            x13_Fault_reset : Bool;
            x14_Setpoint_priority : Bool := TRUE;   // Enabled regardless of the setting of FMOD
            x15_Command_priority : Bool := TRUE;   // Enabled regardless of the setting of CMOD
            x00_Preset_speed_b0 : Bool;
            x01_Preset_speed_b1 : Bool;
            x02_Preset_speed_b2 : Bool;
            x03 : Bool;
            x04_thr2 : Bool;   // THR1 : PT=set value, vL, vb, tHr - THR2 : PT=0, F170, F172, F173
            x05_PI_control : Bool;   // 0:Normal operation, 1:PI OFF
            x06_Acceleration_deceleration_pattern_2 : Bool;   // 0: Acceleration deceleration pattern 1
            x07_DC_braking : Bool;
         END_STRUCT;
         ref : UInt;
      END_STRUCT;
      write2_comm_fault_action : UInt;
      state : USInt;
   END_VAR
   VAR_TEMP
      read6 : Struct   // 16#fe03
         Output_current : UInt;
         Voltage_DC_bus : UInt;
      END_STRUCT;
      u : UInt;
   END_VAR
BEGIN
   // Telemecanique (Schneider) - Altivar 21 inverter
   // VFD (AC-drive)

   (*
   Param:  Name:             Default:    Options:          
   F800    Baud rate         19200       0: 9600 bps, 1: 19200 bps     
   F801    Parity            Even        0: None, 1: Even, 2: Odd      
   F802    Modbus address    1           0 ... 247                     

   CMOD    2 -> Serial communication
   FMOD    4 -> Serial communication
   *)

   "mb_station_block_header"(sb := #sb, mb_query := #mb_query);
   #mb_query.mb_addr := #mb_addr;

   // ==== High priotiry queries =====
   #write1.ref := REAL_TO_UINT(#ref * 100);
   #write1.cmd.x10_Run := #ref <> 0;
   #mb_query(mode := #mb_query.c.write.holding_reg,
             data_addr := 16#fa00,
             data_ptr := #write1);

   // ==== Low priority queries =====
   CASE #state OF
       0:  // Behaviour on modbus fault
           #mb_query(mode := #mb_query.c.write.holding_reg,
                     data_addr := 16#f603,
                     data_ptr := #write2_comm_fault_action);
       1:  // Acceleration time 1  (0.1)
           #u := REAL_TO_UINT(#acceleration_time * 10);
           #mb_query(mode := #mb_query.c.write.holding_reg,
                     data_addr := 16#f603,
                     data_ptr := #u);
       2:  // Basic data, status word
           #mb_query(mode := #mb_query.c.read.holding_reg,
                     data_addr := 16#fd00,
                     data_ptr := #read1);
           IF #mb_query.Done THEN
               #data.Output_frequency :=
               UINT_TO_REAL(#read1.Output_frequency) / 100; // [%]
           END_IF;
       3:  // Where the drive take commands from: modbus or Terminal board.
           #mb_query(mode := #mb_query.c.read.holding_reg,
                     data_addr := 16#fe45,
                     data_ptr := #read2);
       4:  // Alarm word 1
           #mb_query(mode := #mb_query.c.read.holding_reg,
                     data_addr := 16#fe91,
                     data_ptr := #read3_alarm);
       5:  // Alarm word 2
           #mb_query(mode := #mb_query.c.read.holding_reg,
                     data_addr := 16#fe79,
                     data_ptr := #read4_alarm2);
       6:  // Trip code
           #mb_query(mode := #mb_query.c.read.holding_reg,
                     data_addr := 16#fc90,
                     data_ptr := #read5_trip_code);
       7:  // Other data: current, DC-bus
           #mb_query(mode := #mb_query.c.read.holding_reg,
                     data_addr := 16#fe03,
                     data_ptr := #read6);
           IF #mb_query.Done THEN
               #data.Output_current :=
               (* *)UINT_TO_REAL(#read6.Output_current) / 100; // [%]
               #data.Voltage_DC_bus :=
               (* *)UINT_TO_REAL(#read6.Voltage_DC_bus) / 100; // [%]
           END_IF;
       ELSE
           #state += 1;
   END_CASE;
   IF #sb.out.error_comm THEN
       #state := 0;
   ELSIF #mb_query.Done THEN
       #state := SEL(G := #state > 7, IN0 := #state + 1, IN1 := 0);
   END_IF;

   "mb_station_block_footer"(sb := #sb, mb_query := #mb_query);

   (* Trip codes:
   NErr     0  0  No error
   OC1      1  1  Over-current during acceleration
   OC2      2  2  Over-current during deceleration
   OC3      3  3  Over-current during constant speed operation
   OCL      4  4  Over-current in load at startup
   OCA      5  5  Short circuit in arm
   EPHI     8  8  Input phase failure
   EPHO     9  9  Output phase failure
   OP1      A 10 Overvoltage during acceleration
   OP2      B 11 Overvoltage during deceleration
   OP3      C 12 Overvoltage during constant speed operation
   OL1      D 13 Over-LOAD in inverter
   OL2      E 14 Over-LOAD in motor
   OH      10 16 Overheat trip
   E       11 17 Emergency stop
   EEP1    12 18 EEPROM fault 1 (writing error)
   EEP2    13 19 EEPROM fault 2 (reading error)
   EEP3    14 20 EEPROM fault 3 (internal fault)
   Err2    15 21 RAM fault
   Err3    16 22 ROM fault
   Err4    17 23 CPU fault
   Err5    18 24 Communication error trip
   Err7    1A 26 Current detector fault
   Err8    1B 27 Optional circuit board type error
   UC      1D 29 Small-current trip
   UP1     1E 30 Trip due to undervoltage in main circuit
   Ot      20 32 Over-torque trip
   EF2     22 34 Ground fault trip (hardware detection)
   OC1P    25 37 Overcurrent flowing in element during acceleration
   OC2P    26 38 Overcurrent flowing in element during deceleration
   OC3P    27 39 Overcurrent flowing in element during operation
   EtYP    29 41 Inverter type error
   OH2     2E 46 External thermal input
   SOUt    2F 47 VIA cable break
   E-18    32 50 Break in an analog signal cable
   E-19    33 51 CPU fault
   E-20    34 52 Excess torque boost
   E-21    35 53 CPU fault
   Etn1    54 84 Auto-tuning error
   *)
END_FUNCTION_BLOCK

FUNCTION_BLOCK "Schneider_conzerv_EM6430"   // FB91, SCL
{ S7_Optimized_Access := 'TRUE' }
VERSION : 0.1
   VAR_INPUT
      mb_addr : USInt;
   END_VAR
   VAR_IN_OUT
      mb_query : "mb_query";
   END_VAR
   VAR
      sb : "mb_station_block_udt";
      read1_common : Struct
         Apparent_power_total : Real;
         Active_power_total : Real;
         Reactive_power_total : Real;
         Power_factor_average : Real;
         Voltage_average_phase_phase : Real;
         Voltage_average_phase_neutral : Real;
         Current_average : Real;
         Frequency : Real;   // Hz
      END_STRUCT;
      read2_phase : Array[1..3] of Struct
         Apparent_power : Real;
         Active_power : Real;
         Reactive_power : Real;
         Power_factor : Real;
         Voltage_phase_phase : Real;
         Voltage_phase_neutral : Real;
         Current : Real;
      END_STRUCT;
      read3_THD : Struct
         Voltage_THD : Array[1..3] of Real;
         Current_THD : Array[1..3] of Real;
      END_STRUCT;
      read4 : Struct
         Forward_apparent_energy : Real;
         Forward_active_energy : Real;
         Forward_reactive_inductive_energy : Real;
         Forward_reactive_capacitive_energy : Real;
         Reverse_apparent_energy : Real;
         Reverse_active_energy : Real;
         Reverse_reactive_inductive_Energy : Real;
         Reverse_reactive_capacitive_Energy : Real;
         Average_load_percentage : Real;
         Percentage_of_phase_load : Array[1..3] of Real;
         "Unbalanced_%load" : Real;
         "Unbalanced_%_voltage" : Real;
      END_STRUCT;
      read5_common_RMS : Struct
         Apparent_power_total : Real;
         Active_power_total : Real;
         Reactive_power_total : Real;
         Power_factor_average : Real;
         Voltage_average_phase_phase : Real;
         Voltage_average_phase_neutral : Real;
         Current_average : Real;
         Frequency : Real;   // Hz
         _ : UDInt;   // Reserved
         Number_of_interruption : UDInt;
      END_STRUCT;
   END_VAR
BEGIN
   // Schneider-electric - Conzerv EM6430 - Power meters
   // NHA12535-03
   // 
   // https://www.schneider-electric.com/resources/sites/SCHNEIDER_ELECTRIC/
   // content/live/FAQS/276000/FA276938/en_US/EM6430_User_Manual_NHA12535-03.pdf

   "mb_station_block_header"(sb := #sb, mb_query := #mb_query);
   #mb_query.mb_addr := #mb_addr; // Device address.

   #mb_query.mode := #mb_query.c.read.holding_reg;
   #mb_query(data_addr := 3901, data_ptr := #read1_common);
   #mb_query(data_addr := 3917, data_ptr := #read2_phase);
   #mb_query(data_addr := 3861, data_ptr := #read3_THD);
   #mb_query(data_addr := 3959, data_ptr := #read4);
   #mb_query(data_addr := 3001, data_ptr := #read5_common_RMS);

   "mb_station_block_footer"(sb := #sb, mb_query := #mb_query);
END_FUNCTION_BLOCK

FUNCTION_BLOCK "Schneider_PM750"   // FB92, SCL
{ S7_Optimized_Access := 'TRUE' }
VERSION : 0.1
   VAR_INPUT
      mb_addr : UInt;
   END_VAR
   VAR_IN_OUT
      mb_query : "mb_query";
   END_VAR
   VAR
      sb : "mb_station_block_udt";
      data1 : Struct
         "Real Energy, Total" : Real;   // kWh
         "Apparent Energy,Tota" : Real;   // kVAh
         "Reactive Energy,Tota" : Real;   // kVARh
         "Real Power, Total" : Real;   // kW
         "Apparent Power, Total" : Real;   // kVA
         "Reactive Power, Total" : Real;   // kVAR
         "Power Factor, Total" : Real;
         "Voltage, L-L, 3PAverage" : Real;   // Volt
         "Voltage, L-N, 3PAverage" : Real;   // Volt
         "Current, 3P Average" : Real;   // Amp
         Frequency : Real;
      END_STRUCT;
      data2 : Struct
         Current : Array[1..3] of Real;
         Current_N : Real;
      END_STRUCT;
      data3 : Struct
         Voltage_L_L : Array[1..3] of Real;   // [V] 1:L1-L2, 2:L2-L3, 3:L3-L1
         Voltage_L_N : Array[1..3] of Real;   // [V]
         "Real Power" : Array[1..3] of Real;   // kW
         "Apparent Power" : Array[1..3] of Real;   // kVA
         "Reactive Power" : Array[1..3] of Real;   // kVAR
      END_STRUCT;
   END_VAR
BEGIN
   // Schneider - Power Meter 750
   // 63230-507-201A1 - 03/2007
   // 
   // Web: https://www.ccontrols.com/support/dp/SchneiderElectricPowerMeter750.pdf

   "mb_station_block_header"(sb := #sb, mb_query := #mb_query);
   #mb_query.mb_addr := #mb_addr;

   #mb_query.mode := #mb_query.c.read.holding_reg;
   #mb_query(data_addr := 1000, data_ptr := #data1);
   #mb_query(data_addr := 1034, data_ptr := #data2);
   #mb_query(data_addr := 1054, data_ptr := #data3);

   "mb_station_block_footer"(sb := #sb, mb_query := #mb_query);
END_FUNCTION_BLOCK

// folder: Library/Modbus/Station blocks/Siemens

FUNCTION_BLOCK "siemens_PAC3200"   // FB8, SCL
{ S7_Optimized_Access := 'TRUE' }
VERSION : 0.1
   VAR_INPUT
      mb_addr : USInt := 1;
   END_VAR
   VAR_IN_OUT
      mb_query : "mb_query";
   END_VAR
   VAR
      sb : "mb_station_block_udt";
      read1 : Struct
         voltage_L_n : Array[1..3] of Real;
         "voltage _L_L" : Array[1..3] of Real;   // 1:Va-b, 2:Vb-c, 3:Vc-a,
         current : Array[1..3] of Real;
         apparent_power : Array[1..3] of Real;
         active_power : Array[1..3] of Real;
         reactive_power : Array[1..3] of Real;
         power_factor : Array[1..3] of Real;
         THD_R_voltage : Array[1..3] of Real;
      END_STRUCT;
      read2 : Struct
         frequency : Real;   // unit: hz
         avg_voltage_Vph_n : Real;   // unit: V
         avg_voltage_Vph_ph : Real;   // unit: V
         avg_current : Real;   // unit: A
         total_apparent_power : Real;   // unit: VA
         total_active_power : Real;   // unit: W
      END_STRUCT;
      read3 : Struct
         serial_number : String[16];
      END_STRUCT;
   END_VAR
BEGIN
   // - Siemens - PAC3200 - Power meter
   // - http://w3.siemens.com.br/buildingtechnologies/br/
   //   documents/manual-sentron-pac3200.pdf
   //   3.9.3, page 40

   "mb_station_block_header"(sb := #sb, mb_query := #mb_query);
   #mb_query.mb_addr := #mb_addr; // Device address.

   // Tree queries, reading one section of holding registers each.
   #mb_query.mode := #mb_query.c.read.holding_reg;
   #mb_query(data_addr := 1, data_ptr := #read1);
   #mb_query(data_addr := 55, data_ptr := #read2);
   #mb_query(data_addr := 64012, data_ptr := #read3);

   // - Each query reading one section of holding registers.
   // - Data length is automatically calculated for holding and
   //   input regisers.

   "mb_station_block_footer"(sb := #sb, mb_query := #mb_query);
END_FUNCTION_BLOCK

FUNCTION_BLOCK "Siemens_7SR11_7SR12_argus"   // FB53, SCL
{ S7_Optimized_Access := 'TRUE' }
VERSION : 0.1
   VAR_INPUT
      mb_addr : USInt := 1;
   END_VAR
   VAR_OUTPUT
      out1 : Struct
         primary_Voltage_L_L : Array[1..3] of Real;
         primary_Voltage_L_N : Array[1..3] of Real;
         secondary_Voltage_L_N : Array[1..3] of Real;
      END_STRUCT;
      out2 : Struct
         nominal_voltage_degrees_L_L : Array[1..3] of Real;
         nominal_voltage_degrees_L_N : Array[1..3] of Real;
         Vzps : Real;
         Vpps : Real;
         Vnps : Real;
         Vzps_degree : Real;
         Vpps_degree : Real;
         Vnps_degree : Real;
         frequency : Real;
      END_STRUCT;
      out3 : Struct
         primary_current : Array[1..3] of Real;
         secondary_current : Array[1..3] of Real;
         nominal_current : Array[1..3] of Real;
         nominal_current_degrees : Array[1..3] of Real;
         primary_In : Real;
         secondary_In : Real;
         nominal_In : Real;
         primary_Ig : Real;
         secondary_Ig : Real;
         nominal_Ig : Real;
         nominal_Izps : Real;
         nominal_Ipps : Real;
         nominal_Inps : Real;
         nominal_Izps_degrees : Real;
         nominal_Ipps_degrees : Real;
         nominal_Inps_degrees : Real;
      END_STRUCT;
      out4 : Struct
         active_power : Array[1..3] of Real;
         active_power_tot : Real;
         reactive_power : Array[1..3] of Real;
         reactive_power_tot : Real;
         apparent_power : Array[1..3] of Real;
         apparent_power_tot : Real;
         power_factor : Array[1..3] of Real;
         power_factor_tot : Real;
      END_STRUCT;
   END_VAR
   VAR_IN_OUT
      mb_query : "mb_query";
   END_VAR
   VAR
      sb : "mb_station_block_udt";
      out5 : Struct
         act_energy_exp : UDInt;
         act_energy_imp : UDInt;
         react_energy_exp : UDInt;
         react_energy_imp : UDInt;
         thermal_status_Ph_A : UInt;
         thermal_status_Ph_B : UInt;
         thermal_Status_Ph_C : UInt;
      END_STRUCT;
      out6 : Struct
         fault_records : Real;
         event_records : Real;
         waveform_records : Real;
         secondary_voltage : Array[1..3] of Real;
      END_STRUCT;
   END_VAR
   VAR_TEMP
      c : Int;
      read1 : Struct
         primary_Voltage_L_L : Array[1..3] of UDInt;
         primary_Voltage_L_N : Array[1..3] of UDInt;
         secondary_Voltage_L_N : Array[1..3] of UDInt;
      END_STRUCT;
      read2 : Struct
         nominal_voltage_degrees_L_L : Array[1..3] of UDInt;
         nominal_voltage_degrees_L_N : Array[1..3] of UDInt;
         Vzps : UDInt;
         Vpps : UDInt;
         Vnps : UDInt;
         Vzps_degree : UDInt;
         Vpps_degree : UDInt;
         Vnps_degree : UDInt;
         frequency : UDInt;
      END_STRUCT;
      read3 : Struct
         primary_current : Array[1..3] of UDInt;
         secondary_current : Array[1..3] of UDInt;
         nominal_current : Array[1..3] of UDInt;
         nominal_current_degrees : Array[1..3] of UDInt;
         primary_In : UDInt;
         secondary_In : UDInt;
         nominal_In : UDInt;
         primary_Ig : UDInt;
         secondary_Ig : UDInt;
         nominal_Ig : UDInt;
         nominal_Izps : UDInt;
         nominal_Ipps : UDInt;
         nominal_Inps : UDInt;
         nominal_Izps_degrees : UDInt;
         nominal_Ipps_degrees : UDInt;
         nominal_Inps_degrees : UDInt;
      END_STRUCT;
      read4 : Struct
         active_power : Array[1..3] of UDInt;
         active_power_tot : UDInt;
         reactive_power : Array[1..3] of UDInt;
         reactive_power_tot : UDInt;
         apparent_power : Array[1..3] of UDInt;
         apparent_power_tot : UDInt;
         power_factor : Array[1..3] of UDInt;
         power_factor_tot : UDInt;
      END_STRUCT;
      read6 : Struct
         fault_records : UDInt;
         event_records : UDInt;
         waveform_Records : UDInt;
         secondary_voltage : Array[1..3] of UDInt;
      END_STRUCT;
   END_VAR
BEGIN
   // Siemens - 7SR11 & 7SR12 - Argus - Overcurrent Relay
   // Energy Management
   //  
   // - https://cache.industry.siemens.com/dl/files/284/109747284/
   //   att_928907/v1/7SR12_Argus_Complete_Technical_Manual.pdf
   //   ==> page 212  

   "mb_station_block_header"(sb := #sb,
                             mb_query := #mb_query);
   #mb_query.mb_addr := #mb_addr;

   #mb_query.mode := #mb_query.c.mode.read;

   #mb_query(data_addr := 40010,
             data_ptr := #read1);
   IF #mb_query.Done THEN
       FOR #c := 1 TO 3 DO
           #out1.primary_Voltage_L_L[#c] := UDINT_TO_REAL(#read1.primary_Voltage_L_L[#c]) / 1000;
           #out1.primary_Voltage_L_N[#c] := UDINT_TO_REAL(#read1.primary_Voltage_L_N[#c]) / 1000;
           #out1.secondary_Voltage_L_N[#c] := UDINT_TO_REAL(#read1.secondary_Voltage_L_N[#c]) / 1000;
       END_FOR;
   END_IF;

   #mb_query(data_addr := 40034,
             data_ptr := #read2);
   IF #mb_query.Done THEN
       FOR #c := 1 TO 3 DO
           #out2.nominal_voltage_degrees_L_L[#c] := UDINT_TO_REAL(#read2.nominal_voltage_degrees_L_L[#c]) / 1000;
           #out2.nominal_voltage_degrees_L_N[#c] := UDINT_TO_REAL(#read2.nominal_voltage_degrees_L_N[#c]) / 1000;
       END_FOR;
       #out2.Vzps := UDINT_TO_REAL(#read2.Vzps) / 1000;
       #out2.Vpps := UDINT_TO_REAL(#read2.Vpps) / 1000;
       #out2.Vnps := UDINT_TO_REAL(#read2.Vnps) / 1000;
       #out2.Vzps_degree := UDINT_TO_REAL(#read2.Vzps_degree) / 1000;
       #out2.Vpps_degree := UDINT_TO_REAL(#read2.Vpps_degree) / 1000;
       #out2.Vnps_degree := UDINT_TO_REAL(#read2.Vnps_degree) / 1000;
       #out2.frequency := UDINT_TO_REAL(#read2.frequency) / 1000;
   END_IF;

   #mb_query(data_addr := 40064,
             data_ptr := #read3);
   IF #mb_query.Done THEN
       FOR #c := 1 TO 3 DO
           #out3.primary_current[#c] := UDINT_TO_REAL(#read3.primary_current[#c]) / 1000;
           #out3.secondary_current[#c] := UDINT_TO_REAL(#read3.secondary_current[#c]) / 1000;
           #out3.nominal_current[#c] := UDINT_TO_REAL(#read3.nominal_current[#c]) / 1000;
           #out3.nominal_current_degrees[#c] := UDINT_TO_REAL(#read3.nominal_current_degrees[#c]) / 1000;
       END_FOR;
       #out3.primary_In := UDINT_TO_REAL(#read3.primary_In) / 1000;
       #out3.secondary_In := UDINT_TO_REAL(#read3.secondary_In) / 1000;
       #out3.nominal_In := UDINT_TO_REAL(#read3.nominal_In) / 1000;
       #out3.primary_Ig := UDINT_TO_REAL(#read3.primary_Ig) / 1000;
       #out3.secondary_Ig := UDINT_TO_REAL(#read3.secondary_Ig) / 1000;
       #out3.nominal_Ig := UDINT_TO_REAL(#read3.nominal_Ig) / 1000;
       #out3.nominal_Izps := UDINT_TO_REAL(#read3.nominal_Izps) / 1000;
       #out3.nominal_Ipps := UDINT_TO_REAL(#read3.nominal_Ipps) / 1000;
       #out3.nominal_Inps := UDINT_TO_REAL(#read3.nominal_Inps) / 1000;
       #out3.nominal_Izps_degrees := UDINT_TO_REAL(#read3.nominal_Izps_degrees) / 1000;
       #out3.nominal_Ipps_degrees := UDINT_TO_REAL(#read3.nominal_Ipps_degrees) / 1000;
       #out3.nominal_Inps_degrees := UDINT_TO_REAL(#read3.nominal_Inps_degrees) / 1000;
   END_IF;

   #mb_query(data_addr := 40112,
             data_ptr := #read4);
   IF #mb_query.Done THEN
       FOR #c := 1 TO 3 DO
           #out4.active_power[#c] := UDINT_TO_REAL(#read4.active_power[#c]) / 1000;
           #out4.reactive_power[#c] := UDINT_TO_REAL(#read4.reactive_power[#c]) / 1000;
           #out4.apparent_power[#c] := UDINT_TO_REAL(#read4.apparent_power[#c]) / 1000;
           #out4.power_factor[#c] := UDINT_TO_REAL(#read4.power_factor[#c]) / 1000;
       END_FOR;
       #out4.active_power_tot := UDINT_TO_REAL(#read4.active_power_tot) / 1000;
       #out4.reactive_power_tot := UDINT_TO_REAL(#read4.reactive_power_tot) / 1000;
       #out4.apparent_power_tot := UDINT_TO_REAL(#read4.apparent_power_tot) / 1000;
       #out4.power_factor_tot := UDINT_TO_REAL(#read4.power_factor_tot) / 1000;
   END_IF;

   #mb_query(data_addr := 40144,
             data_ptr := #out5);

   #mb_query(data_addr := 40167,
             data_ptr := #read6);
   IF #mb_query.Done THEN
       FOR #c := 1 TO 3 DO
           #out6.secondary_voltage[#c] := UDINT_TO_REAL(#read6.secondary_voltage[#c]) / 1000;
       END_FOR;
       #out6.fault_records := UDINT_TO_REAL(#read6.fault_records) / 1000;
       #out6.event_records := UDINT_TO_REAL(#read6.event_records) / 1000;
       #out6.waveform_records := UDINT_TO_REAL(#read6.waveform_Records) / 1000;
   END_IF;

   "mb_station_block_footer"(sb := #sb,
                             mb_query := #mb_query);
END_FUNCTION_BLOCK

FUNCTION_BLOCK "Siemens_MAG_6000"   // FB54, SCL
{ S7_Optimized_Access := 'TRUE' }
VERSION : 0.1
   VAR_INPUT
      mb_addr : UInt;
   END_VAR
   VAR_IN_OUT
      mb_query : "mb_query";
   END_VAR
   VAR
      sb : "mb_station_block_udt";
      flow : Struct
         velocity : Real;   // mm/s
         flow : Real;
      END_STRUCT;
      totalizer : Array[1..3] of UDInt;
   END_VAR
BEGIN
   // Siemens - SITRANS F M MAG 6000

   "mb_station_block_header"(sb := #sb, mb_query := #mb_query);
   #mb_query.mb_addr := #mb_addr;

   #mb_query.mode := #mb_query.c.read.holding_reg;
   #mb_query(data_addr := 2999, data_ptr := #flow);
   #mb_query(data_addr := 3016, data_ptr := #totalizer);

   "mb_station_block_footer"(sb := #sb, mb_query := #mb_query);
END_FUNCTION_BLOCK

FUNCTION_BLOCK "Siemens_MASS_6000"   // FB55, SCL
{ S7_Optimized_Access := 'TRUE' }
VERSION : 0.1
   VAR_INPUT
      mb_addr : UInt;
   END_VAR
   VAR_IN_OUT
      mb_query : "mb_query";
   END_VAR
   VAR
      sb : "mb_station_block_udt";
      flow : Struct
         massflow : Real;   // [kg/s]
         volumeflow : Real;   // [m3/s]
         density : Real;   // [kg/m3]
         temperature : Real;   // [Â°C]
         fraction : Array[1..2] of Real;   // [kg/s]
         "%_fraction" : Real;   // [%]
         totalizer_1 : Array[1..2] of UDInt;   // [kg or m3]
         totalizer_2 : Array[1..2] of UDInt;   // [kg or m3]
         totalizer_real : Array[1..2] of Real;   // [kg or m3]
      END_STRUCT;
   END_VAR
BEGIN
   // Siemens - MASS 6000
   // https://cache.industry.siemens.com/dl/files/906/44880906/
   // att_70364/v1/USMII_MODBUS_AOM_OI_En_en-US.pdf

   "mb_station_block_header"(sb := #sb, mb_query := #mb_query);
   #mb_query.mb_addr := #mb_addr;

   #mb_query.mode := #mb_query.c.read.holding_reg;
   #mb_query(data_addr := 3000, data_ptr := #flow);

   "mb_station_block_footer"(sb := #sb, mb_query := #mb_query);
END_FUNCTION_BLOCK

FUNCTION_BLOCK "Siemens_sed2_modbus2"   // FB57, SCL
{ S7_Optimized_Access := 'TRUE' }
VERSION : 0.1
   VAR_INPUT
      mb_addr : UInt;
      ref : Real;   // 0-100% ( -100% reverse)
   END_VAR
   VAR_OUTPUT
      speed : Real;   // rpm
      current : Real;   // A x10
      torque : Real;   // Nm x10
      actual_pwr : Real;   // kW x100
      total_kwh : Real;   // kWh
      dc_bus_volt : Real;   // V
   END_VAR
   VAR_IN_OUT
      mb_query : "mb_query";
   END_VAR
   VAR
      sb : "mb_station_block_udt";
      write1 : Struct
         wdog_time : UInt := 1500;   // [ms]
         wdog_action : Word := 1;   // 1:stop, 0:no action
         freq_ref : UInt;
         run_enable : UInt;
         reverse : UInt;
         cmd_start : UInt;
         fault_ack : UInt;
      END_STRUCT;
      write2 : Struct
         current_limit : UInt := 4000;   // A x0
         accel_time : UInt := 1000;   // s x100
         decel_time : UInt := 1000;   // s x100
         manual : UInt;
      END_STRUCT;
      write3 : Struct
         freq_max : UInt := 5000;   // HZ x100
      END_STRUCT;
      read1 : Struct
         freq_output : UInt;   // Hz x10
         speed : UInt;   // rpm
         current : UInt;   // A x10
         torque : UInt;   // Nm x10
         actual_pwr : UInt;   // kW x100
         total_kwh : UInt;   // kWh
         dc_bus_volt : UInt;   // V
         reference : UInt;   // Hz x10
         rated_pwr : UInt;   // kWx100
         output_volts : UInt;
         reverse : UInt;
         run : UInt;
         at_max_freq : UInt;
         ctrl_mode : UInt;   // 1:SERIAL, 0:LOCAL
         enabled : UInt;
         ready_to_run : UInt;
         analog_in_1 : UInt;
         analog_in_2 : UInt;
      END_STRUCT;
      read2 : Struct
         digital_in : Array[1..6] of UInt;
         fault : UInt;
         last_fault : UInt;
         fault_hist : Array[1..4] of UInt;
         warning : UInt;
         last_warning : UInt;
      END_STRUCT;
   END_VAR
   VAR_TEMP
      "real" : Real;
   END_VAR
BEGIN
   // Siemens - SED2-MODBUS2 - Variable Frequency Drive
   // Modbus RTU Interface Module for SED2 
   // 
   // https://www.downloads.siemens.com/download-center/
   // Download.aspx?pos=download&fct=getasset&id1=A6V10073869

   #write1.reverse := BOOL_TO_UINT(#ref < 0);
   #"real" := NORM_X(MIN := 0, VALUE := #ref, MAX := ABS(100));
   #write1.freq_ref := SCALE_X(MIN := 0, VALUE := #"real", MAX := 16#4000);
   #write1.run_enable := BOOL_TO_UINT(#ref <> 0);
   #write1.cmd_start := BOOL_TO_UINT(#ref <> 0);

   "mb_station_block_header"(sb := #sb,
                             mb_query := #mb_query);
   #mb_query.mb_addr := #mb_addr;

   #mb_query.mode := #mb_query.c.mode.write;
   #mb_query(data_addr := 40001,
             data_ptr := #write1);
   #mb_query(data_addr := 40010,
             data_ptr := #write2);
   #mb_query(data_addr := 40016,
             data_ptr := #write3);

   #mb_query.mode := #mb_query.c.mode.read;
   #mb_query(data_addr := 40024,
             data_ptr := #read1);
   #mb_query(data_addr := 40048,
             data_ptr := #read2);

   "mb_station_block_footer"(sb := #sb,
                             mb_query := #mb_query);

   #speed := UINT_TO_REAL(#read1.speed);
   #current := UINT_TO_REAL(#read1.current) / 10;
   #torque := UINT_TO_REAL(#read1.torque) / 10;
   #actual_pwr := UINT_TO_REAL(#read1.actual_pwr) / 100;
   #total_kwh := UINT_TO_REAL(#read1.total_kwh);
   #dc_bus_volt := UINT_TO_REAL(#read1.dc_bus_volt);
END_FUNCTION_BLOCK

FUNCTION_BLOCK "Siemens_Sinamics_G120"   // FB58, SCL
{ S7_Optimized_Access := 'TRUE' }
VERSION : 0.1
   VAR_INPUT
      mb_addr : UInt;
      ref : Real;
   END_VAR
   VAR_IN_OUT
      mb_query : "mb_query";
   END_VAR
   VAR
      sb : "mb_station_block_udt";
      read : Struct
         stw : Struct
            x08_Speed_setpoint : Bool;   // Actual value deviation within tolerance t_off
            x09_Control_requested : Bool;
            x10_f_or_n_comparison_value_reached_exceeded : Bool;
            x11_I_M_or_P_limit_not_reached : Bool;
            x12 : Bool;
            x13_No_motor_overtemperature_alarm : Bool;
            x14_Motor_rotates_forwards : Bool;   // 0 = Motor rotates backwards (n_act < 0)
            x15_No_alarm_thermal_overload_power_unit : Bool;
            x00_Ready_to_power_up : Bool;
            x01_Ready_to_operate : Bool;   // (DC link loaded, pulses blocked)
            x02_Operation_enabled : Bool;   // (drive follows n_set)
            x03_Fault_present : Bool;
            x04_No_coast_down_active : Bool;   // (OFF2 inactive)
            x05_No_fast_stop_active : Bool;   // (OFF3 inactive)
            x06_power_on_inhibit_active : Bool;
            x07_Alarm_present : Bool;
         END_STRUCT;
         actual : Int;
      END_STRUCT;
      write : Struct
         ctw : Struct
            x08 : Bool;
            x09 : Bool;
            x10_control_via_PLC : Bool := TRUE;
            x11_reversal : Bool;
            x12 : Bool;
            x13_Motorized_potentiometer_setpoint_raise : Bool;
            x14_Motorized_potentiometer_setpoint_lower : Bool;
            x15 : Bool;
            x00_R_TRIG_ON : Bool;   // 0 = OFF1 (braking with ramp-function generator, then pulse cancllation &ready-to-power-up)
            x01_No_OFF2 : Bool := TRUE;   // enable is possible. 0 = OFF2 (immediate pulse cancellation and power-on inhibit)
            x02_No_OFF3 : Bool := TRUE;   // enable is possible. 0 = OFF3 braking with the OFF3 ramp p1135, then pulse cancellation andpower-on inhibit)
            x03_Enable_operation : Bool := TRUE;   // (pulses can be enabled) 0 = Inhibit operation (cancel pulses)
            x04_Operating_condition : Bool;   // (the ramp-function generator can be enabled)0 = Inhibit ramp-function generator (set the ramp-function generator output tozero)
            x05_Enable_the_ramp_function_generator : Bool;   // 0 = Stop the ramp-function generator (freeze the ramp-function generatoroutput)
            x06_enable_setpoint : Bool := TRUE;   // 0 = Inhibit setpoint (set the ramp-function generator input to zero)
            x07_R_TRIG_acknowledge_faults : Bool;
         END_STRUCT;
         setpoint : Int;
      END_STRUCT;
   END_VAR
BEGIN
   // Siemens - SINAMICS G120
   // 
   // Web: https://cache.industry.siemens.com/dl/files/944/
   // 35928944/att_7966/v1/application_cu230_modbus_v1_2_en.pdf

   "mb_station_block_header"(sb := #sb, mb_query := #mb_query);
   #mb_query.mb_addr := #mb_addr;

   #mb_query.mode := #mb_query.c.read.holding_reg;
   #mb_query(data_addr := 40110, data_ptr := #read);

   #write.ctw.x00_R_TRIG_ON :=
   (* *)#ref <> 0
   (* *)AND NOT #read.stw.x07_Alarm_present
   (* *)AND #read.stw.x01_Ready_to_operate
   (* *)AND #read.stw.x00_Ready_to_power_up;
   #write.setpoint := REAL_TO_INT(#ref);

   #mb_query.mode := #mb_query.c.write.holding_reg;
   #mb_query(data_addr := 40100, data_ptr := #write);

   "mb_station_block_footer"(sb := #sb, mb_query := #mb_query);
END_FUNCTION_BLOCK

FUNCTION_BLOCK "Siemens_SITRANS_F_M_MAG_8000"   // FB59, SCL
{ S7_Optimized_Access := 'TRUE' }
VERSION : 0.1
   VAR_INPUT
      mb_addr : UInt;
   END_VAR
   VAR_IN_OUT
      mb_query : "mb_query";
   END_VAR
   VAR
      sb : "mb_station_block_udt";
      flow : Struct
         velocity : Real;   // mm/s
         flow : Real;
      END_STRUCT;
      totalizer : Array[1..3] of UDInt;
   END_VAR
BEGIN
   // Siemens - SITRANS F M MAG 8000
   // https://cache.industry.siemens.com/dl/files/509/54091509/
   // att_100244/v1/A5E03409989_01_MAG8000_MODBUS_AOM_OI_.pdf

   "mb_station_block_header"(sb := #sb, mb_query := #mb_query);
   #mb_query.mb_addr := #mb_addr;

   #mb_query.mode := #mb_query.c.read.holding_reg;
   #mb_query(data_addr := 2999, data_ptr := #flow);
   #mb_query(data_addr := 3016, data_ptr := #totalizer);

   "mb_station_block_footer"(sb := #sb, mb_query := #mb_query);
END_FUNCTION_BLOCK

FUNCTION_BLOCK "Siemens_vav_compact_controller"   // FB60, SCL
{ S7_Optimized_Access := 'TRUE' }
VERSION : 0.1
   VAR_INPUT
      mb_addr : UInt;
      sp : Real;   // setpoint
      sp_backup : Real;
   END_VAR
   VAR_IN_OUT
      mb_query : "mb_query";
   END_VAR
   VAR
      sb : "mb_station_block_udt";
      read : Struct
         Actual_position : Int;
         Actual_Flow_rel : UInt;
         Actual_Flow_abs : UInt;
         Actual_Pressure : UInt;
      END_STRUCT;
      write1 : Struct
         Setpoint : Int;
      END_STRUCT;
      write2 : Struct
         backup_mode : Int;
         backup_position : Int;
      END_STRUCT;
   END_VAR
BEGIN
   // Siemens - VAV compact controller 
   // GDB181.1E/MO Operating voltage AC 24 V, 5 Nm
   // GLB181.1E/MO Operating voltage AC 24 V, 10 Nm

   // https://www.micromatic.no/globalassets/inriver/resources/
   // bruksanvisning_ko1320-28.pdf

   "mb_station_block_header"(sb := #sb, mb_query := #mb_query);
   #mb_query.mb_addr := #mb_addr;

   #mb_query.mode := #mb_query.c.read.holding_reg;
   #mb_query(data_addr := 3, data_ptr := #read);

   #mb_query.mode := #mb_query.c.write.holding_reg;
   #write1.Setpoint := REAL_TO_INT(#sp) * 100;
   #mb_query(data_addr := 1, data_ptr := #write1);
   #write2.backup_position := REAL_TO_INT(#sp_backup) * 100;
   #mb_query(data_addr := 513, data_ptr := #write2);

   "mb_station_block_footer"(sb := #sb, mb_query := #mb_query);

   (*
   Backup mode (write 2)
   0 = Go to BackupPosition
   1 = Keep last position
   2 = Disabled
   *)
END_FUNCTION_BLOCK

FUNCTION_BLOCK "Siemens_SIWAREX_WP251"   // FB93, SCL
{ S7_Optimized_Access := 'TRUE' }
VERSION : 0.1
   VAR_INPUT
      mb_addr : UInt;
   END_VAR
   VAR_IN_OUT
      mb_query : "mb_query";
   END_VAR
   VAR
      sb : "mb_station_block_udt";
      read1 : Struct
         Unit_of_weight : UInt;   // x1000
         Gross_identifier : UInt;
         Code_for_regulations : UInt;
         Reserve : UInt;
         weighing_range_min : UInt;
         weighing_range_max : Real;
         Calibration_weight : Array[0..2] of Real;
         Calibration_digits : Array[0..2] of Real;
         Scale_interval : Array[0..2] of Real;   // (Page 64)
      END_STRUCT;
      read2 : Struct
         stat : Struct
            x08 : Bool;
            x09 : Bool;
            x10 : Bool;
            x11 : Bool;
            x12 : Bool;
            x13 : Bool;
            x14 : Bool;
            x15 : Bool;
            x00 : Bool;
            x01 : Bool;
            x02 : Bool;
            x03 : Bool;
            x04 : Bool;
            x05 : Bool;
            x06 : Bool;
            x07 : Bool;
         END_STRUCT;
         Reserve : UInt;
         Max_tare_load : Real;
         Max_negative_zero_limit_power_on : Real;
         Max_positive_zero_limit_power_on : Real;
         Max_negative_zero_limit_semi_automatically : Real;
         Max_positive_zero_limit_semi_automatically : Real;
      END_STRUCT;
      read3 : Struct
         standstill : Array[1..2] of Struct
            range : Real;
            "time" : Time;
            max_waiting_time : Time;
         END_STRUCT;
         frequency_low_pass_filter1 : Real;
         Order_no_low_pass_filter1 : UInt;
         depth_average_filter : UInt;
         reserve_1 : UInt;
         weighing_operating_mode : UInt;
         resolution_of_master_totalizer : Real;
         Reserve_2 : Real;
         SecureDisplay_including_weighing_range_data : UInt;
      END_STRUCT;
      read4 : Struct
         SecureDisplay_interface : UInt;   // (Page 71)
         String_header_version_SecureDisplay : String[2];
         SecureDisplay_version : String[12];
         Minimum_zoom_factor_of_SecureDisplay : UInt;
         Reserve_1 : Array[1..3] of Real;
         Reserve_2 : Array[1..3] of UInt;
         Grid_frequency : UInt;   // 0: 50 Hz, 1: 60Hz
      END_STRUCT;
      write1 : Struct
         Smallest_weight_below_TU2 : Real;
         Highest_weight_above_TH2 : Real;
         Single_setpoin : Real;
         Net_weight_average_value : Real;
         Standard_deviation : Real;
      END_STRUCT;
   END_VAR
BEGIN
   // Siemens - SIWAREX WP251 - Electronic Weighing System
   // A5E37203357A
   // 
   // https://cache.industry.siemens.com/dl/files/751/109481751/att_893477/v1/Manual_SIWAREX_WP251_en_en-US.pdf

   "mb_station_block_header"(sb := #sb, mb_query := #mb_query);
   #mb_query.mb_addr := #mb_addr;

   #mb_query.mode := #mb_query.c.read.holding_reg;
   #mb_query(data_addr := 1011, data_ptr := #read1);
   #mb_query(data_addr := 1032, data_ptr := #read2);
   #mb_query(data_addr := 1044, data_ptr := #read3);
   #mb_query(data_addr := 1067, data_ptr := #read4);

   #mb_query.mode := #mb_query.c.write.holding_reg;
   #mb_query(data_addr := 4101, data_ptr := #write1);

   "mb_station_block_footer"(sb := #sb, mb_query := #mb_query);

   (*
   Unit of weight:
   0: "mg"
   1: "g"
   2: "kg"
   3: "t"
   4: "oz" (ounce)
   5: "lb" (pound)
   6: "T" (=short tons)
   7: "TL" (= long tons)

   Gross identifier:
   0: "brutto" 
   1: "Gross"

   Code for regulations:
   0: None
   1: OIML

   Weighing operating mode (Page 71):
   0: NAWI – Filling
   1: NAWI – Removal
   10: AWI
   20: ACI – Filling 
   21: ACI – Removal

   *)
END_FUNCTION_BLOCK

// folder: Library/Modbus/Station blocks/Swan

FUNCTION_BLOCK "Swan_AMI_CACE"   // FB65, SCL
{ S7_Optimized_Access := 'TRUE' }
VERSION : 0.1
   VAR_INPUT
      mb_addr : USInt;
   END_VAR
   VAR_IN_OUT
      mb_query : "mb_query";
   END_VAR
   VAR
      sb : "mb_station_block_udt";
      data : Struct
         cond_sc : Array[1..3] of Real;   // µS
         Temp : Array[1..3] of Real;
         flow : Real;
         pH : Real;
         alkalyzer : Real;
         cond_uc : Array[1..3] of Real;
         Pt1000_Temp : Array[1..3] of Real;
         raw_flow : Real;
         case_temperature : Real;
         EDI_voltage : Real;
         EDI_current : Real;
         Degasser_temperature : Real;
         Degasser_boiling_point : Real;
         Degasser_PWM : Real;
         Degasser_line_voltage : Real;
         Degasser_air_pressure : Real;
         Degasser_Case_Temp : Real;
         signal_output : Array[1..2] of Real;
         "Instrument Display Status" : DWord;
      END_STRUCT;
      alarm : Struct
         x00_Cond_1_Alarm_high : Bool;
         x01_Cond_1_Alarm_low : Bool;
         x02_Cond_2_Alarm_high : Bool;
         x03_Cond_2_Alarm_low : Bool;
         x04_Cond_3_Alarm_high : Bool;
         x05_Cond_3_Alarm_low : Bool;
         x06_Temp_1_high : Bool;
         x07_Temp_1_low : Bool;
         x08_sample_flow_high : Bool;
         x09_sample_flow_low : Bool;
         x10_temp_1_shorted : Bool;
         x11_temp_1_disconnected : Bool;
         x12_case_temp_high : Bool;
         x13_case_temp_low : Bool;
         x14_pH_Error : Bool;
         x15_Degasser_frontend : Bool;
         x16_control_timeout : Bool;
         x17_Degasser_disconnected : Bool;
         x18_Temp_2_shorted : Bool;
         x19_Temp_2_disconnected : Bool;
         x20_Temp_3_shorted : Bool;
         x21_Temp_3_disconnected : Bool;
         x22_Degasser_Ctl_Timeout : Bool;
         x23_Input_Active : Bool;
         x24_IC_MK41T56 : Bool;
         x25_IC_LM75 : Bool;
         x26_IC_PCF8574 : Bool;
         x27_Signal_output_open : Bool;
         x28_Calibration_Degasser : Bool;
         x29_EEprom_Front_end : Bool;
         x30_Calibration_Recout : Bool;
         x31_Wrong_Front_end : Bool;
         x32_pH_Alarm_high : Bool;
         x33_pH_Alarm_low : Bool;
         x34_Alkali_Alarm_high : Bool;
         x35_Alkali_Alarm_low : Bool;
         x36_Temp_2_high : Bool;
         x37_Temp_2_low : Bool;
         x38_Temp_3_high : Bool;
         x39_Temp_3_low : Bool;
         x40_Degasser_Line_Voltage : Bool;
         x41_Degasser_Temperature : Bool;
         x42_EDI_out_of_range : Bool;
         x43_No_sample_flow : Bool;
         x44_EDI_DAC_disconnected : Bool;
         "x45_ EDI_ADC_disconnected" : Bool;
         x46 : Bool;
         x47_EDI_module_exhausted : Bool;
      END_STRUCT;
      write : Struct
         x0_relay_contacts_1 : Bool;
         x1_relay_contacts_2 : Bool;
         x2 : Bool;
         x3 : Bool;
         x4 : Bool;
         x5 : Bool;
         x6 : Bool;
         x7 : Bool;
      END_STRUCT;
   END_VAR
BEGIN
   // Swan - AMI CACE - Conductivity measurement 
   // Swan analytical instruments
   // http://www.swan.ch/GetAttachment.axd?attaName=e82f8e94-ab32-4930-8c9d-a56dc0847f61
   // Page 9

   "mb_station_block_header"(sb := #sb,
                             mb_query := #mb_query);
   #mb_query.mb_addr := #mb_addr;
   #mb_query.data_addr := 0;

   #mb_query(mode := #mb_query.c.read.input_reg,
             data_ptr := #data);

   #mb_query(mode := #mb_query.c.read.discrete_input,
             data_ptr := #alarm);

   (*#mb_query(mode := #mb_query.c.write.discrete_output,
             data_len := 2,
             data_ptr := #write);*)

   "mb_station_block_footer"(sb := #sb,
                             mb_query := #mb_query);
END_FUNCTION_BLOCK

FUNCTION_BLOCK "Swan_AMI_Codes-II_CC"   // FB66, SCL
{ S7_Optimized_Access := 'TRUE' }
VERSION : 0.1
   VAR_INPUT
      mb_addr : USInt;
   END_VAR
   VAR_IN_OUT
      mb_query : "mb_query";
   END_VAR
   VAR
      sb : "mb_station_block_udt";
      data : Struct
         free_available_chlorine : Real;   // ppm
         total_chlorine_1_tc1 : Real;   // ppm
         total_chlorine_2_tc2 : Real;   // ppm
         calculated_monochloramine : Real;   // ppm
         calculated_combined_chlorine : Real;   // ppm
         calculated_dichloramine : Real;   // ppm
         temperature : Real;   // °C
         flow : Real;   // B/s
         pH : Real;   // pH
         absorbance : Real;
         photometer_frequency : Real;   // Hz
         remaining_DPD_buffer : Real;   // %
         remaining_potassium_Iodide : Real;   // %
         remaining_cleaning_solution : Real;   // %
         raw_temp_NTK5 : Real;   // Ohm
         raw_flow : Real;   // Hz
         raw_pH : Real;   // mV
         case_temperature : Real;   // °C
         signal_output_1 : Real;   // mA
         signal_output_2 : Real;   // mA
         instrument_display_status : Real;
      END_STRUCT;
      alarm : Struct
         x00_high_fac : Bool;
         x01_low_fac : Bool;
         x02_high_tc1 : Bool;
         x03_low_tc1 : Bool;
         x04_high_tc2 : Bool;
         x05_low_tc2 : Bool;
         x06_sample_temp_high : Bool;
         x07_sample_temp_low : Bool;
         x08_sample_flow_high : Bool;
         x09_sample_flow_low : Bool;
         x10_Temp_shorted : Bool;
         x11_Temp_disconnected : Bool;
         x12_case_temp_high : Bool;
         x13_case_temp_low : Bool;
         x14_valve_1_defective : Bool;
         x15_dis_invalid : Bool;
         x16_control_timeout : Bool;
         x17_reagent_pump : Bool;
         x18_photometer_not_connected : Bool;
         x19_photometer_dirty : Bool;
         x20_absorbance_too_high : Bool;
         x21_reagent_empty : Bool;
         x22_cleaning_reagent : Bool;
         x23_input_active : Bool;
         x24_IC_MK41T56 : Bool;
         x25_IC_LM75 : Bool;
         x26_IC_PCF8574 : Bool;
         x27_signal_output_open : Bool;
         x28_EEprom_motherboard : Bool;
         x29_EEprom_front_end : Bool;
         x30_calibration_recout : Bool;
         x31_wrong_front_end : Bool;
         x32_high_cmc : Bool;
         x33_low_cmc : Bool;
         x34_high_ccc : Bool;
         x35_low_ccc : Bool;
         x36_high_cdc : Bool;
         x37_low_cdc : Bool;
         x38_high_pH : Bool;
         x39_low_pH : Bool;
         x40_DPD_buffer : Bool;
         x41_potassium_Iodide : Bool;
         x42_cleaning_solution : Bool;
         x43 : Bool;
         x44 : Bool;
         x45 : Bool;
         x46 : Bool;
         x47 : Bool;
      END_STRUCT;
      write : Struct
         x0_relay_contacts_1 : Bool;
         x1_relay_contacts_2 : Bool;
         x2_hold : Bool;
         x3_Remote_off : Bool;
         x4 : Bool;
         x5 : Bool;
         x6 : Bool;
         x7 : Bool;
      END_STRUCT;
   END_VAR
BEGIN
   // Swan - AMI Codes-II CC
   //
   // http://www.swan.ch/GetAttachment.axd?attaName=e82f8e94-ab32-4930-8c9d-a56dc0847f61
   // Page 17

   "mb_station_block_header"(sb := #sb,
                             mb_query := #mb_query);
   #mb_query.mb_addr := #mb_addr;
   #mb_query.data_addr := 0;

   #mb_query(mode := #mb_query.c.read.input_reg,
             data_ptr := #data);

   #mb_query(mode := #mb_query.c.read.discrete_input,
             data_ptr := #alarm);

   (*#mb_query(mode := #mb_query.c.write.discrete_output,
             data_len := 4,
             data_ptr := #write);*)

   "mb_station_block_footer"(sb := #sb,
                             mb_query := #mb_query);
END_FUNCTION_BLOCK

FUNCTION_BLOCK "Swan_AMI_Hydrogen"   // FB67, SCL
{ S7_Optimized_Access := 'TRUE' }
VERSION : 0.1
   VAR_INPUT
      mb_addr : USInt;
   END_VAR
   VAR_IN_OUT
      mb_query : "mb_query";
   END_VAR
   VAR
      sb : "mb_station_block_udt";
      data : Struct
         hydrogen : Real;   // ppb
         temperature : Real;   // °C
         flow : Real;   // l/h
         saturation : Real;   // %
         air_pressure : Real;   // hPa
         raw_Current_temp_compensated : Real;   // nA
         raw_current_uncompensated : Real;   // nA
         raw_temp_Pt1000 : Real;   // Ω
         raw_flow : Real;   // Hz
         reserved : Real;
         case_temperature : Real;   // °C
         signal_output_1 : Real;   // mA
         signal_output_2 : Real;   // mA
         instrument_display_status : UDInt;
      END_STRUCT;
      alarm : Struct
         x00_hydrogen_alarm_high : Bool;
         x01_hydrogen_alarm_low : Bool;
         x02_saturation_alarm_high : Bool;
         x03_saturation_alarm_low : Bool;
         x04 : Bool;
         x05 : Bool;
         x06_sample_temp_high : Bool;
         x07_sample_temp_low : Bool;
         x08_sample_flow_high : Bool;
         x09_sample_flow_low : Bool;
         x10_temp_shorted : Bool;
         x11_temp_disconnected : Bool;
         x12_case_temp_high : Bool;
         x13_case_temp_low : Bool;
         x14 : Bool;
         x15 : Bool;
         x16_control_timeout : Bool;
         x17_faraday_efficiency_QED : Bool;
         x18_quality_assurance : Bool;
         x19 : Bool;
         x20 : Bool;
         x21 : Bool;
         x22 : Bool;
         x23_input_active : Bool;
         x24_IC_MK41T56 : Bool;
         x25_IC_LM75 : Bool;
         x26_IC_PCF8574 : Bool;
         x27_Signal_output_open : Bool;
         x28_EEprom_Motherboard : Bool;
         x29_EEprom_Front_end : Bool;
         x30_Calibration_Recout : Bool;
         x31_Wrong_Front_end : Bool;
         x32 : Bool;
         x33 : Bool;
         x34 : Bool;
         x35 : Bool;
         x36 : Bool;
         x37 : Bool;
         x38 : Bool;
         x39 : Bool;
         x40 : Bool;
         x41 : Bool;
         x42 : Bool;
         x43 : Bool;
         x44 : Bool;
         x45 : Bool;
         x46 : Bool;
         x47_Status_Electrolyte_depleted : Bool;
      END_STRUCT;
      write : Struct
         x0_relay_contacts_1 : Bool;
         x1_relay_contacts_2 : Bool;
         x2_hold : Bool;
         x3_Remote_off : Bool;
         x4 : Bool;
         x5 : Bool;
         x6 : Bool;
         x7 : Bool;
      END_STRUCT;
   END_VAR
BEGIN
   // Swan - AMI Hydrogen
   // Swan analytical instruments
   // http://www.swan.ch/GetAttachment.axd?attaName=e82f8e94-ab32-4930-8c9d-a56dc0847f61
   // Page 37

   "mb_station_block_header"(sb := #sb,
                             mb_query := #mb_query);
   #mb_query.mb_addr := #mb_addr;
   #mb_query.data_addr := 0;

   #mb_query(mode := #mb_query.c.read.input_reg,
             data_ptr := #data);

   #mb_query(mode := #mb_query.c.read.discrete_input,
             data_ptr := #alarm);

   (*#mb_query(mode := #mb_query.c.write.discrete_output,
             data_len := 4,
             data_ptr := #write);*)

   "mb_station_block_footer"(sb := #sb,
                             mb_query := #mb_query);
END_FUNCTION_BLOCK

FUNCTION_BLOCK "Swan_AMI_Oxysafe"   // FB68, SCL
{ S7_Optimized_Access := 'TRUE' }
VERSION : 0.1
   VAR_INPUT
      mb_addr : USInt;
   END_VAR
   VAR_IN_OUT
      mb_query : "mb_query";
   END_VAR
   VAR
      sb : "mb_station_block_udt";
      data : Struct
         oxygen : Real;   // ppm
         temperature : Real;   // °C
         flow : Real;   // l/h
         saturation : Real;   // %
         air_pressure : Real;   // hPa
         raw_Oxygen_temp_compensated : Real;   // nA
         raw_oxygen_temp_uncompensated : Real;   // nA
         raw_Temp_Pt1000 : Real;   // Ohm
         raw_flow : Real;   // Hz
         remaining_electrolyte : Real;   // %
         case_temperature : Real;   // °C
         signal_output_1 : Real;   // mA
         signal_output_2 : Real;   // mA
         instrument_display_status : DWord;
      END_STRUCT;
      alarm : Struct
         x00_Oxygen_alarm_high : Bool;
         x01_Oxygen_alarm_low : Bool;
         x02_Saturation_alarm_high : Bool;
         x03_Saturation_alarm_low : Bool;
         x04 : Bool;
         x05 : Bool;
         x06_Sample_temp_high : Bool;
         x07_Sample_temp_low : Bool;
         x08_sample_flow_high : Bool;
         x09_sample_flow_low : Bool;
         x10_temp_shorted : Bool;
         x11_temp_disconnected : Bool;
         x12_case_temp_high : Bool;
         x13_case_temp_low : Bool;
         x14 : Bool;
         x15 : Bool;
         x16_control_timeout : Bool;
         x17_Faraday_efficiency_QED : Bool;
         x18 : Bool;
         x19 : Bool;
         x20 : Bool;
         x21 : Bool;
         x22 : Bool;
         x23_input_active : Bool;
         x24_IC_MK41T56 : Bool;
         x25_IC_LM75 : Bool;
         x26_IC_PCF8574 : Bool;
         x27_Signal_output_open : Bool;
         x28_EEprom_Motherboard : Bool;
         x29_EEprom_Front_end : Bool;
         x30_Calibration_Recout : Bool;
         x31_Wrong_Front_end : Bool;
         x32 : Bool;
         x33 : Bool;
         x34 : Bool;
         x35 : Bool;
         x36 : Bool;
         x37 : Bool;
         x38 : Bool;
         x39 : Bool;
         x40_Electrolyte_depleted : Bool;
         x41 : Bool;
         x42 : Bool;
         x43 : Bool;
         x44 : Bool;
         x45 : Bool;
         x46 : Bool;
         x47 : Bool;
      END_STRUCT;
      write : Struct
         x0_relay_contacts_1 : Bool;
         x1_relay_contacts_2 : Bool;
         x2_hold : Bool;
         x3_Remote_off : Bool;
         x4 : Bool;
         x5 : Bool;
         x6 : Bool;
         x7 : Bool;
      END_STRUCT;
   END_VAR
BEGIN
   // Swan - AMI - Oxysafe
   // Swan analytical instruments
   // http://www.swan.ch/GetAttachment.axd?attaName=e82f8e94-ab32-4930-8c9d-a56dc0847f61
   // Page 53

   "mb_station_block_header"(sb := #sb,
                             mb_query := #mb_query);
   #mb_query.mb_addr := #mb_addr;
   #mb_query.data_addr := 0;

   #mb_query(mode := #mb_query.c.read.input_reg,
             data_ptr := #data);

   #mb_query(mode := #mb_query.c.read.discrete_input,
             data_ptr := #alarm);

   (*#mb_query(mode := #mb_query.c.write.discrete_output,
             data_len := 4,
             data_ptr := #write);*) 

   "mb_station_block_footer"(sb := #sb,
                             mb_query := #mb_query);
END_FUNCTION_BLOCK

